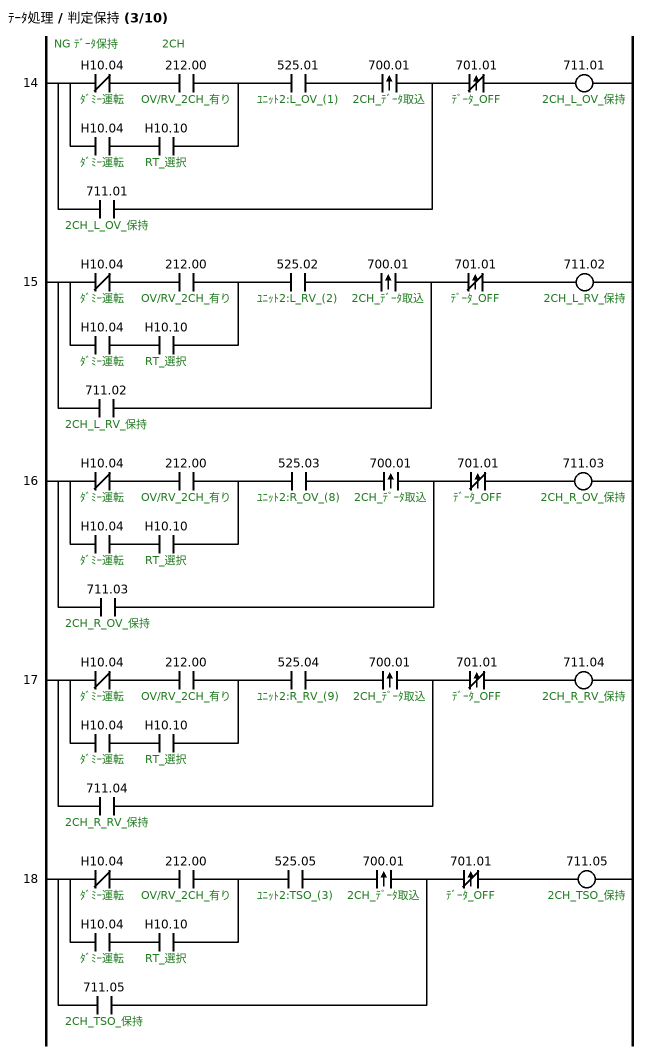
; [picture p144: ﾃｰﾀ処理 / 判定保持, rungs 14-18]
; rung 14: NG ﾃﾞｰﾀ保持　　　　2CH
LDNOT H10.04  ; ﾀﾞﾐｰ運転
AND 212.00  ; OV/RV_2CH_有り
LD H10.04  ; ﾀﾞﾐｰ運転
AND H10.10  ; RT_選択
ORLD
AND 525.01  ; ﾕﾆｯﾄ2:L_OV_(1)
@AND 700.01  ; 2CH_ﾃﾞｰﾀ取込
OR 711.01  ; 2CH_L_OV_保持
@ANDNOT 701.01  ; ﾃﾞｰﾀ_OFF
OUT 711.01  ; 2CH_L_OV_保持
; rung 15
LDNOT H10.04  ; ﾀﾞﾐｰ運転
AND 212.00  ; OV/RV_2CH_有り
LD H10.04  ; ﾀﾞﾐｰ運転
AND H10.10  ; RT_選択
ORLD
AND 525.02  ; ﾕﾆｯﾄ2:L_RV_(2)
@AND 700.01  ; 2CH_ﾃﾞｰﾀ取込
OR 711.02  ; 2CH_L_RV_保持
@ANDNOT 701.01  ; ﾃﾞｰﾀ_OFF
OUT 711.02  ; 2CH_L_RV_保持
; rung 16
LDNOT H10.04  ; ﾀﾞﾐｰ運転
AND 212.00  ; OV/RV_2CH_有り
LD H10.04  ; ﾀﾞﾐｰ運転
AND H10.10  ; RT_選択
ORLD
AND 525.03  ; ﾕﾆｯﾄ2:R_OV_(8)
@AND 700.01  ; 2CH_ﾃﾞｰﾀ取込
OR 711.03  ; 2CH_R_OV_保持
@ANDNOT 701.01  ; ﾃﾞｰﾀ_OFF
OUT 711.03  ; 2CH_R_OV_保持
; rung 17
LDNOT H10.04  ; ﾀﾞﾐｰ運転
AND 212.00  ; OV/RV_2CH_有り
LD H10.04  ; ﾀﾞﾐｰ運転
AND H10.10  ; RT_選択
ORLD
AND 525.04  ; ﾕﾆｯﾄ2:R_RV_(9)
@AND 700.01  ; 2CH_ﾃﾞｰﾀ取込
OR 711.04  ; 2CH_R_RV_保持
@ANDNOT 701.01  ; ﾃﾞｰﾀ_OFF
OUT 711.04  ; 2CH_R_RV_保持
; rung 18
LDNOT H10.04  ; ﾀﾞﾐｰ運転
AND 212.00  ; OV/RV_2CH_有り
LD H10.04  ; ﾀﾞﾐｰ運転
AND H10.10  ; RT_選択
ORLD
AND 525.05  ; ﾕﾆｯﾄ2:TSO_(3)
@AND 700.01  ; 2CH_ﾃﾞｰﾀ取込
OR 711.05  ; 2CH_TSO_保持
@ANDNOT 701.01  ; ﾃﾞｰﾀ_OFF
OUT 711.05  ; 2CH_TSO_保持

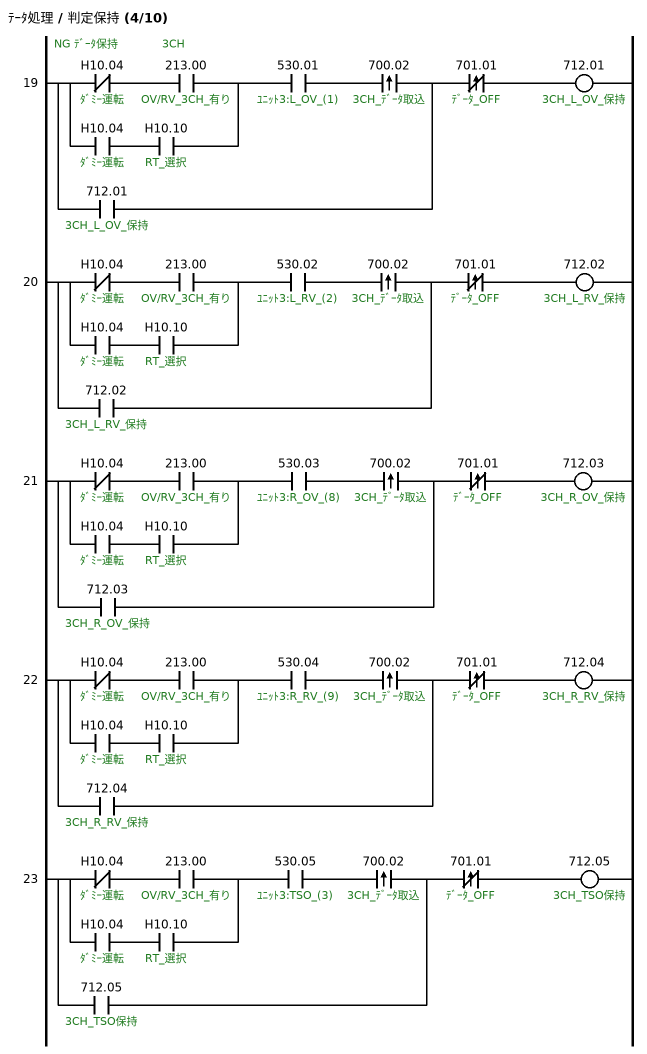
; rung 19: NG ﾃﾞｰﾀ保持　　　　3CH
LDNOT H10.04  ; ﾀﾞﾐｰ運転
AND 213.00  ; OV/RV_3CH_有り
LD H10.04  ; ﾀﾞﾐｰ運転
AND H10.10  ; RT_選択
ORLD
AND 530.01  ; ﾕﾆｯﾄ3:L_OV_(1)
@AND 700.02  ; 3CH_ﾃﾞｰﾀ取込
OR 712.01  ; 3CH_L_OV_保持
@ANDNOT 701.01  ; ﾃﾞｰﾀ_OFF
OUT 712.01  ; 3CH_L_OV_保持
; rung 20
LDNOT H10.04  ; ﾀﾞﾐｰ運転
AND 213.00  ; OV/RV_3CH_有り
LD H10.04  ; ﾀﾞﾐｰ運転
AND H10.10  ; RT_選択
ORLD
AND 530.02  ; ﾕﾆｯﾄ3:L_RV_(2)
@AND 700.02  ; 3CH_ﾃﾞｰﾀ取込
OR 712.02  ; 3CH_L_RV_保持
@ANDNOT 701.01  ; ﾃﾞｰﾀ_OFF
OUT 712.02  ; 3CH_L_RV_保持
; rung 21
LDNOT H10.04  ; ﾀﾞﾐｰ運転
AND 213.00  ; OV/RV_3CH_有り
LD H10.04  ; ﾀﾞﾐｰ運転
AND H10.10  ; RT_選択
ORLD
AND 530.03  ; ﾕﾆｯﾄ3:R_OV_(8)
@AND 700.02  ; 3CH_ﾃﾞｰﾀ取込
OR 712.03  ; 3CH_R_OV_保持
@ANDNOT 701.01  ; ﾃﾞｰﾀ_OFF
OUT 712.03  ; 3CH_R_OV_保持
; rung 22
LDNOT H10.04  ; ﾀﾞﾐｰ運転
AND 213.00  ; OV/RV_3CH_有り
LD H10.04  ; ﾀﾞﾐｰ運転
AND H10.10  ; RT_選択
ORLD
AND 530.04  ; ﾕﾆｯﾄ3:R_RV_(9)
@AND 700.02  ; 3CH_ﾃﾞｰﾀ取込
OR 712.04  ; 3CH_R_RV_保持
@ANDNOT 701.01  ; ﾃﾞｰﾀ_OFF
OUT 712.04  ; 3CH_R_RV_保持
; rung 23
LDNOT H10.04  ; ﾀﾞﾐｰ運転
AND 213.00  ; OV/RV_3CH_有り
LD H10.04  ; ﾀﾞﾐｰ運転
AND H10.10  ; RT_選択
ORLD
AND 530.05  ; ﾕﾆｯﾄ3:TSO_(3)
@AND 700.02  ; 3CH_ﾃﾞｰﾀ取込
OR 712.05  ; 3CH_TSO保持
@ANDNOT 701.01  ; ﾃﾞｰﾀ_OFF
OUT 712.05  ; 3CH_TSO保持

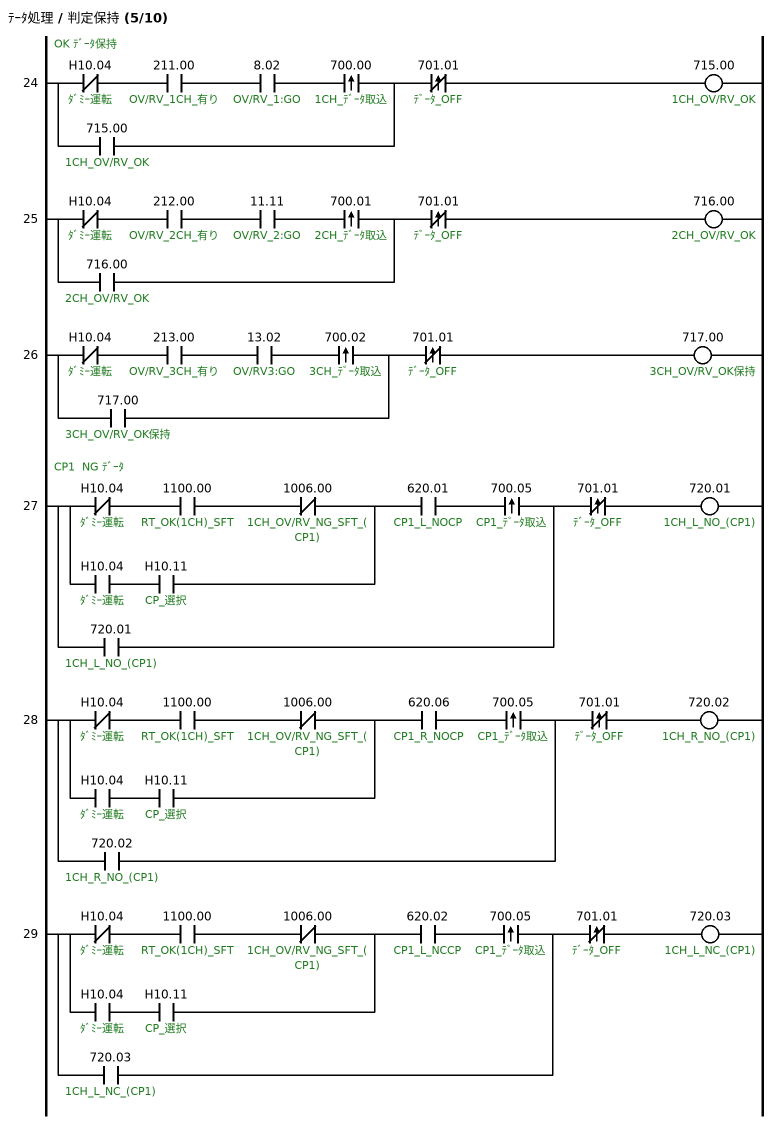
; rung 24: OK ﾃﾞｰﾀ保持
LDNOT H10.04  ; ﾀﾞﾐｰ運転
AND 211.00  ; OV/RV_1CH_有り
AND 8.02  ; OV/RV_1:GO
@AND 700.00  ; 1CH_ﾃﾞｰﾀ取込
OR 715.00  ; 1CH_OV/RV_OK
@ANDNOT 701.01  ; ﾃﾞｰﾀ_OFF
OUT 715.00  ; 1CH_OV/RV_OK
; rung 25
LDNOT H10.04  ; ﾀﾞﾐｰ運転
AND 212.00  ; OV/RV_2CH_有り
AND 11.11  ; OV/RV_2:GO
@AND 700.01  ; 2CH_ﾃﾞｰﾀ取込
OR 716.00  ; 2CH_OV/RV_OK
@ANDNOT 701.01  ; ﾃﾞｰﾀ_OFF
OUT 716.00  ; 2CH_OV/RV_OK
; rung 26
LDNOT H10.04  ; ﾀﾞﾐｰ運転
AND 213.00  ; OV/RV_3CH_有り
AND 13.02  ; OV/RV3:GO
@AND 700.02  ; 3CH_ﾃﾞｰﾀ取込
OR 717.00  ; 3CH_OV/RV_OK保持
@ANDNOT 701.01  ; ﾃﾞｰﾀ_OFF
OUT 717.00  ; 3CH_OV/RV_OK保持
; rung 27: CP1  NG ﾃﾞｰﾀ
LDNOT H10.04  ; ﾀﾞﾐｰ運転
AND 1100.00  ; RT_OK(1CH)_SFT
ANDNOT 1006.00  ; 1CH_OV/RV_NG_SFT_(CP1)
LD H10.04  ; ﾀﾞﾐｰ運転
AND H10.11  ; CP_選択
ORLD
AND 620.01  ; CP1_L_NOCP
@AND 700.05  ; CP1_ﾃﾞｰﾀ取込
OR 720.01  ; 1CH_L_NO_(CP1)
@ANDNOT 701.01  ; ﾃﾞｰﾀ_OFF
OUT 720.01  ; 1CH_L_NO_(CP1)
; rung 28
LDNOT H10.04  ; ﾀﾞﾐｰ運転
AND 1100.00  ; RT_OK(1CH)_SFT
ANDNOT 1006.00  ; 1CH_OV/RV_NG_SFT_(CP1)
LD H10.04  ; ﾀﾞﾐｰ運転
AND H10.11  ; CP_選択
ORLD
AND 620.06  ; CP1_R_NOCP
@AND 700.05  ; CP1_ﾃﾞｰﾀ取込
OR 720.02  ; 1CH_R_NO_(CP1)
@ANDNOT 701.01  ; ﾃﾞｰﾀ_OFF
OUT 720.02  ; 1CH_R_NO_(CP1)
; rung 29
LDNOT H10.04  ; ﾀﾞﾐｰ運転
AND 1100.00  ; RT_OK(1CH)_SFT
ANDNOT 1006.00  ; 1CH_OV/RV_NG_SFT_(CP1)
LD H10.04  ; ﾀﾞﾐｰ運転
AND H10.11  ; CP_選択
ORLD
AND 620.02  ; CP1_L_NCCP
@AND 700.05  ; CP1_ﾃﾞｰﾀ取込
OR 720.03  ; 1CH_L_NC_(CP1)
@ANDNOT 701.01  ; ﾃﾞｰﾀ_OFF
OUT 720.03  ; 1CH_L_NC_(CP1)

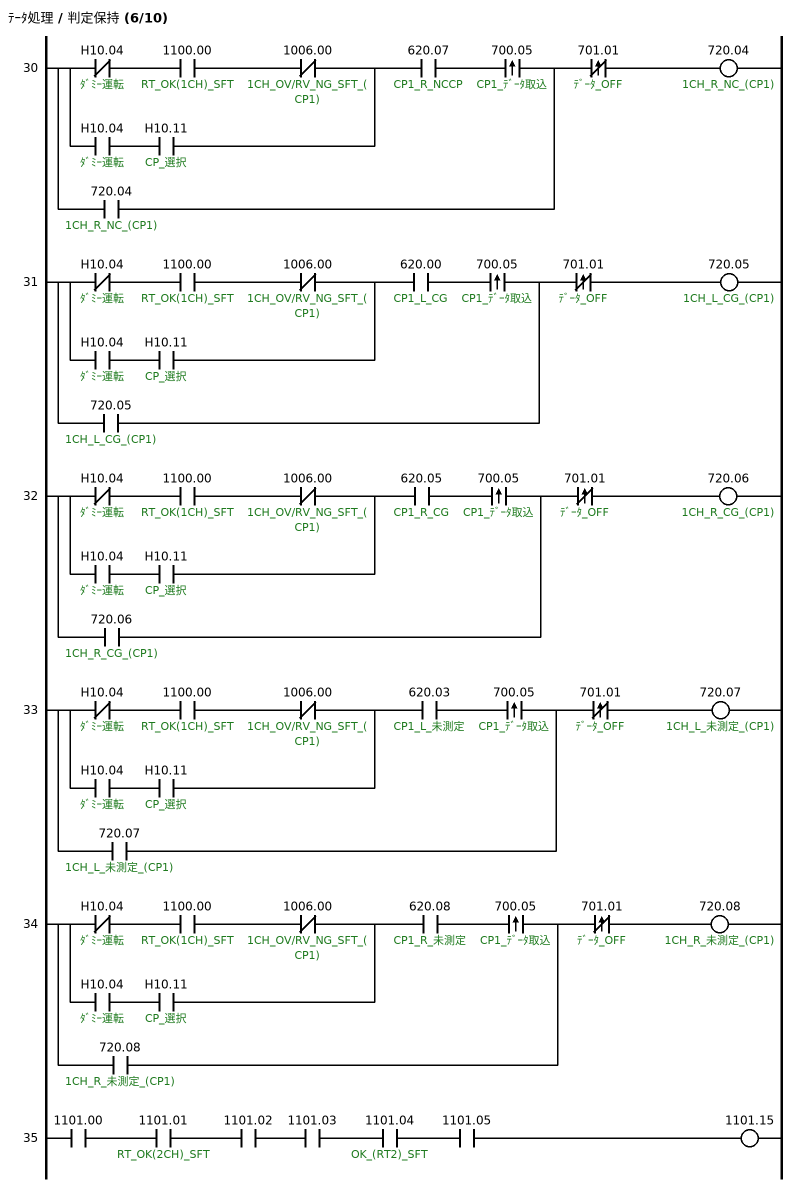
; rung 30
LDNOT H10.04  ; ﾀﾞﾐｰ運転
AND 1100.00  ; RT_OK(1CH)_SFT
ANDNOT 1006.00  ; 1CH_OV/RV_NG_SFT_(CP1)
LD H10.04  ; ﾀﾞﾐｰ運転
AND H10.11  ; CP_選択
ORLD
AND 620.07  ; CP1_R_NCCP
@AND 700.05  ; CP1_ﾃﾞｰﾀ取込
OR 720.04  ; 1CH_R_NC_(CP1)
@ANDNOT 701.01  ; ﾃﾞｰﾀ_OFF
OUT 720.04  ; 1CH_R_NC_(CP1)
; rung 31
LDNOT H10.04  ; ﾀﾞﾐｰ運転
AND 1100.00  ; RT_OK(1CH)_SFT
ANDNOT 1006.00  ; 1CH_OV/RV_NG_SFT_(CP1)
LD H10.04  ; ﾀﾞﾐｰ運転
AND H10.11  ; CP_選択
ORLD
AND 620.00  ; CP1_L_CG
@AND 700.05  ; CP1_ﾃﾞｰﾀ取込
OR 720.05  ; 1CH_L_CG_(CP1)
@ANDNOT 701.01  ; ﾃﾞｰﾀ_OFF
OUT 720.05  ; 1CH_L_CG_(CP1)
; rung 32
LDNOT H10.04  ; ﾀﾞﾐｰ運転
AND 1100.00  ; RT_OK(1CH)_SFT
ANDNOT 1006.00  ; 1CH_OV/RV_NG_SFT_(CP1)
LD H10.04  ; ﾀﾞﾐｰ運転
AND H10.11  ; CP_選択
ORLD
AND 620.05  ; CP1_R_CG
@AND 700.05  ; CP1_ﾃﾞｰﾀ取込
OR 720.06  ; 1CH_R_CG_(CP1)
@ANDNOT 701.01  ; ﾃﾞｰﾀ_OFF
OUT 720.06  ; 1CH_R_CG_(CP1)
; rung 33
LDNOT H10.04  ; ﾀﾞﾐｰ運転
AND 1100.00  ; RT_OK(1CH)_SFT
ANDNOT 1006.00  ; 1CH_OV/RV_NG_SFT_(CP1)
LD H10.04  ; ﾀﾞﾐｰ運転
AND H10.11  ; CP_選択
ORLD
AND 620.03  ; CP1_L_未測定
@AND 700.05  ; CP1_ﾃﾞｰﾀ取込
OR 720.07  ; 1CH_L_未測定_(CP1)
@ANDNOT 701.01  ; ﾃﾞｰﾀ_OFF
OUT 720.07  ; 1CH_L_未測定_(CP1)
; rung 34
LDNOT H10.04  ; ﾀﾞﾐｰ運転
AND 1100.00  ; RT_OK(1CH)_SFT
ANDNOT 1006.00  ; 1CH_OV/RV_NG_SFT_(CP1)
LD H10.04  ; ﾀﾞﾐｰ運転
AND H10.11  ; CP_選択
ORLD
AND 620.08  ; CP1_R_未測定
@AND 700.05  ; CP1_ﾃﾞｰﾀ取込
OR 720.08  ; 1CH_R_未測定_(CP1)
@ANDNOT 701.01  ; ﾃﾞｰﾀ_OFF
OUT 720.08  ; 1CH_R_未測定_(CP1)
; rung 35
LD 1101.00
AND 1101.01  ; RT_OK(2CH)_SFT
AND 1101.02
AND 1101.03
AND 1101.04  ; OK_(RT2)_SFT
AND 1101.05
OUT 1101.15

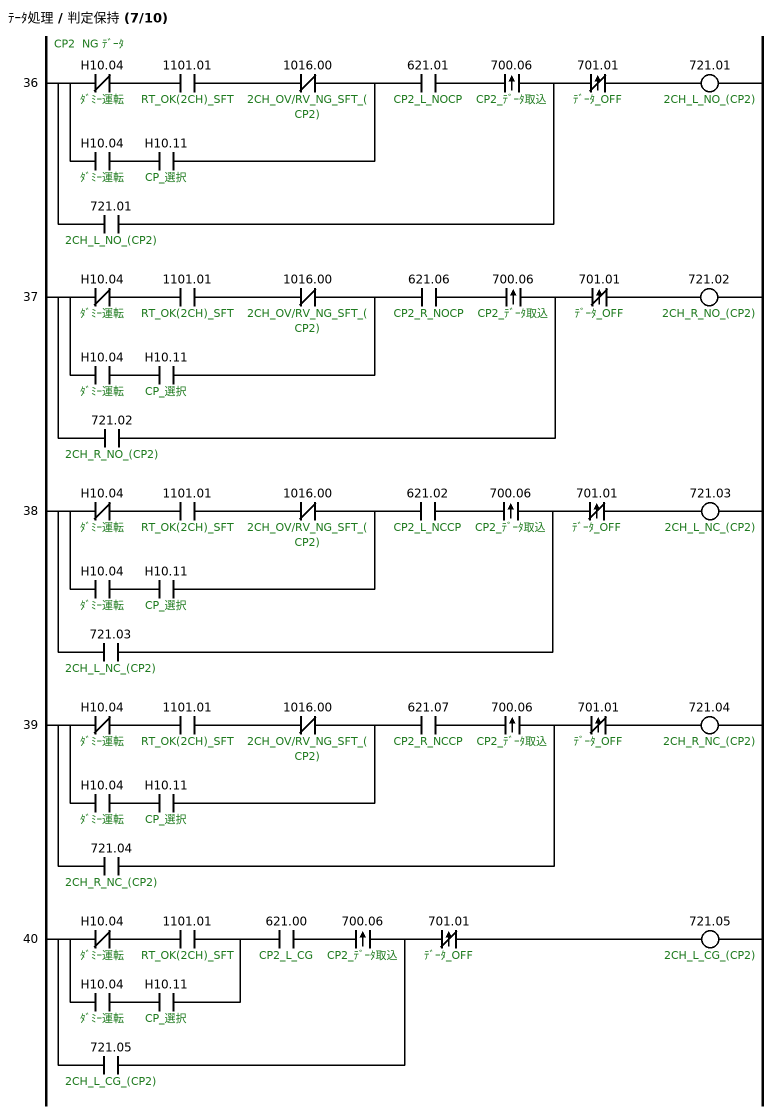
; rung 36: CP2  NG ﾃﾞｰﾀ
LDNOT H10.04  ; ﾀﾞﾐｰ運転
AND 1101.01  ; RT_OK(2CH)_SFT
ANDNOT 1016.00  ; 2CH_OV/RV_NG_SFT_(CP2)
LD H10.04  ; ﾀﾞﾐｰ運転
AND H10.11  ; CP_選択
ORLD
AND 621.01  ; CP2_L_NOCP
@AND 700.06  ; CP2_ﾃﾞｰﾀ取込
OR 721.01  ; 2CH_L_NO_(CP2)
@ANDNOT 701.01  ; ﾃﾞｰﾀ_OFF
OUT 721.01  ; 2CH_L_NO_(CP2)
; rung 37
LDNOT H10.04  ; ﾀﾞﾐｰ運転
AND 1101.01  ; RT_OK(2CH)_SFT
ANDNOT 1016.00  ; 2CH_OV/RV_NG_SFT_(CP2)
LD H10.04  ; ﾀﾞﾐｰ運転
AND H10.11  ; CP_選択
ORLD
AND 621.06  ; CP2_R_NOCP
@AND 700.06  ; CP2_ﾃﾞｰﾀ取込
OR 721.02  ; 2CH_R_NO_(CP2)
@ANDNOT 701.01  ; ﾃﾞｰﾀ_OFF
OUT 721.02  ; 2CH_R_NO_(CP2)
; rung 38
LDNOT H10.04  ; ﾀﾞﾐｰ運転
AND 1101.01  ; RT_OK(2CH)_SFT
ANDNOT 1016.00  ; 2CH_OV/RV_NG_SFT_(CP2)
LD H10.04  ; ﾀﾞﾐｰ運転
AND H10.11  ; CP_選択
ORLD
AND 621.02  ; CP2_L_NCCP
@AND 700.06  ; CP2_ﾃﾞｰﾀ取込
OR 721.03  ; 2CH_L_NC_(CP2)
@ANDNOT 701.01  ; ﾃﾞｰﾀ_OFF
OUT 721.03  ; 2CH_L_NC_(CP2)
; rung 39
LDNOT H10.04  ; ﾀﾞﾐｰ運転
AND 1101.01  ; RT_OK(2CH)_SFT
ANDNOT 1016.00  ; 2CH_OV/RV_NG_SFT_(CP2)
LD H10.04  ; ﾀﾞﾐｰ運転
AND H10.11  ; CP_選択
ORLD
AND 621.07  ; CP2_R_NCCP
@AND 700.06  ; CP2_ﾃﾞｰﾀ取込
OR 721.04  ; 2CH_R_NC_(CP2)
@ANDNOT 701.01  ; ﾃﾞｰﾀ_OFF
OUT 721.04  ; 2CH_R_NC_(CP2)
; rung 40
LDNOT H10.04  ; ﾀﾞﾐｰ運転
AND 1101.01  ; RT_OK(2CH)_SFT
LD H10.04  ; ﾀﾞﾐｰ運転
AND H10.11  ; CP_選択
ORLD
AND 621.00  ; CP2_L_CG
@AND 700.06  ; CP2_ﾃﾞｰﾀ取込
OR 721.05  ; 2CH_L_CG_(CP2)
@ANDNOT 701.01  ; ﾃﾞｰﾀ_OFF
OUT 721.05  ; 2CH_L_CG_(CP2)

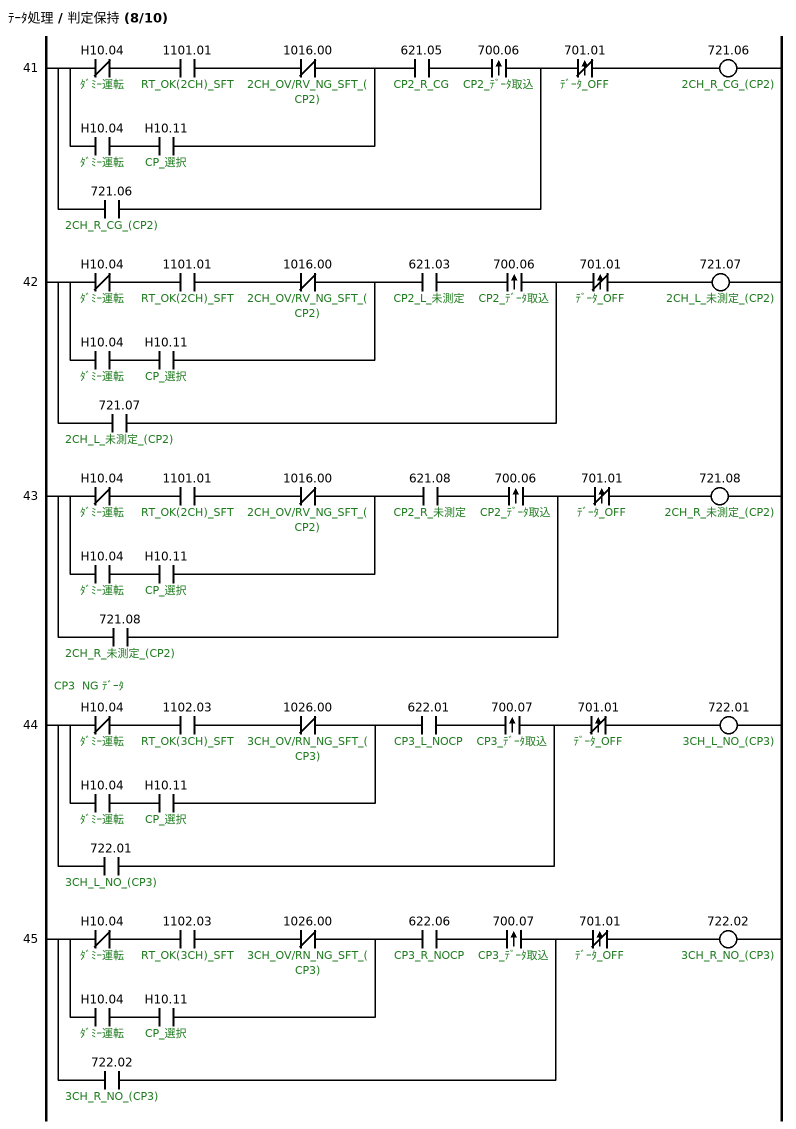
; rung 41
LDNOT H10.04  ; ﾀﾞﾐｰ運転
AND 1101.01  ; RT_OK(2CH)_SFT
ANDNOT 1016.00  ; 2CH_OV/RV_NG_SFT_(CP2)
LD H10.04  ; ﾀﾞﾐｰ運転
AND H10.11  ; CP_選択
ORLD
AND 621.05  ; CP2_R_CG
@AND 700.06  ; CP2_ﾃﾞｰﾀ取込
OR 721.06  ; 2CH_R_CG_(CP2)
@ANDNOT 701.01  ; ﾃﾞｰﾀ_OFF
OUT 721.06  ; 2CH_R_CG_(CP2)
; rung 42
LDNOT H10.04  ; ﾀﾞﾐｰ運転
AND 1101.01  ; RT_OK(2CH)_SFT
ANDNOT 1016.00  ; 2CH_OV/RV_NG_SFT_(CP2)
LD H10.04  ; ﾀﾞﾐｰ運転
AND H10.11  ; CP_選択
ORLD
AND 621.03  ; CP2_L_未測定
@AND 700.06  ; CP2_ﾃﾞｰﾀ取込
OR 721.07  ; 2CH_L_未測定_(CP2)
@ANDNOT 701.01  ; ﾃﾞｰﾀ_OFF
OUT 721.07  ; 2CH_L_未測定_(CP2)
; rung 43
LDNOT H10.04  ; ﾀﾞﾐｰ運転
AND 1101.01  ; RT_OK(2CH)_SFT
ANDNOT 1016.00  ; 2CH_OV/RV_NG_SFT_(CP2)
LD H10.04  ; ﾀﾞﾐｰ運転
AND H10.11  ; CP_選択
ORLD
AND 621.08  ; CP2_R_未測定
@AND 700.06  ; CP2_ﾃﾞｰﾀ取込
OR 721.08  ; 2CH_R_未測定_(CP2)
@ANDNOT 701.01  ; ﾃﾞｰﾀ_OFF
OUT 721.08  ; 2CH_R_未測定_(CP2)
; rung 44: CP3  NG ﾃﾞｰﾀ
LDNOT H10.04  ; ﾀﾞﾐｰ運転
AND 1102.03  ; RT_OK(3CH)_SFT
ANDNOT 1026.00  ; 3CH_OV/RN_NG_SFT_(CP3)
LD H10.04  ; ﾀﾞﾐｰ運転
AND H10.11  ; CP_選択
ORLD
AND 622.01  ; CP3_L_NOCP
@AND 700.07  ; CP3_ﾃﾞｰﾀ取込
OR 722.01  ; 3CH_L_NO_(CP3)
@ANDNOT 701.01  ; ﾃﾞｰﾀ_OFF
OUT 722.01  ; 3CH_L_NO_(CP3)
; rung 45
LDNOT H10.04  ; ﾀﾞﾐｰ運転
AND 1102.03  ; RT_OK(3CH)_SFT
ANDNOT 1026.00  ; 3CH_OV/RN_NG_SFT_(CP3)
LD H10.04  ; ﾀﾞﾐｰ運転
AND H10.11  ; CP_選択
ORLD
AND 622.06  ; CP3_R_NOCP
@AND 700.07  ; CP3_ﾃﾞｰﾀ取込
OR 722.02  ; 3CH_R_NO_(CP3)
@ANDNOT 701.01  ; ﾃﾞｰﾀ_OFF
OUT 722.02  ; 3CH_R_NO_(CP3)

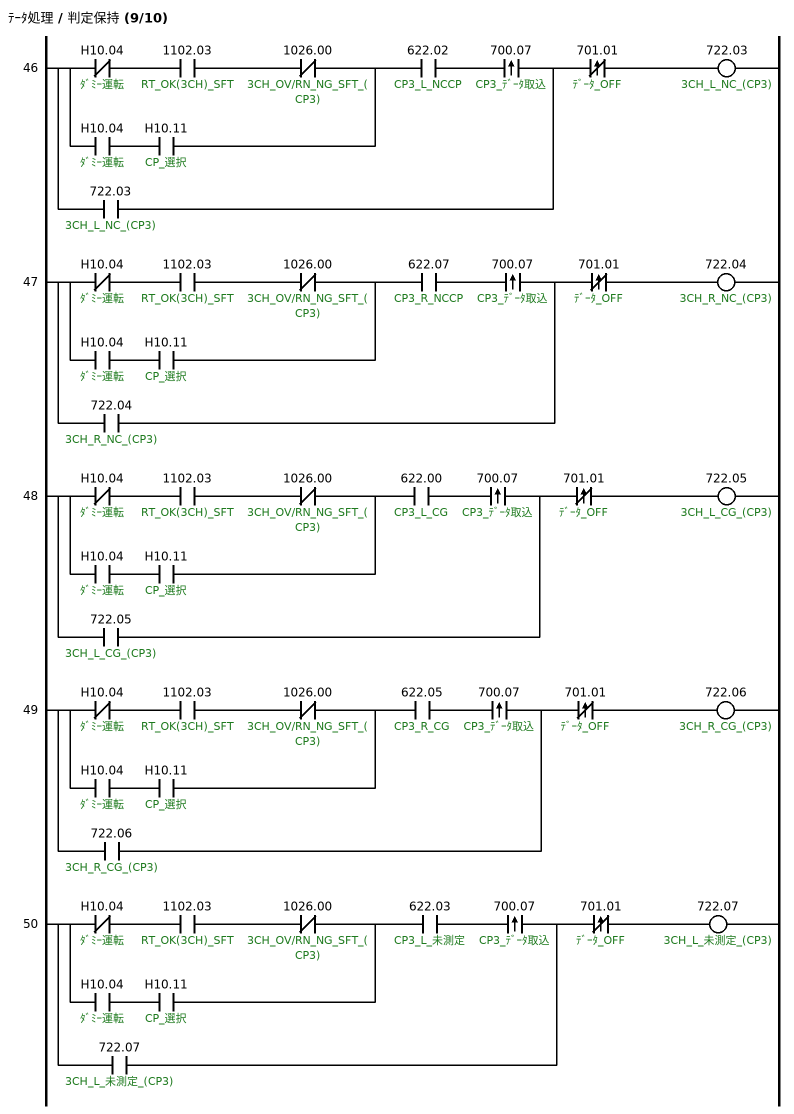
; rung 46
LDNOT H10.04  ; ﾀﾞﾐｰ運転
AND 1102.03  ; RT_OK(3CH)_SFT
ANDNOT 1026.00  ; 3CH_OV/RN_NG_SFT_(CP3)
LD H10.04  ; ﾀﾞﾐｰ運転
AND H10.11  ; CP_選択
ORLD
AND 622.02  ; CP3_L_NCCP
@AND 700.07  ; CP3_ﾃﾞｰﾀ取込
OR 722.03  ; 3CH_L_NC_(CP3)
@ANDNOT 701.01  ; ﾃﾞｰﾀ_OFF
OUT 722.03  ; 3CH_L_NC_(CP3)
; rung 47
LDNOT H10.04  ; ﾀﾞﾐｰ運転
AND 1102.03  ; RT_OK(3CH)_SFT
ANDNOT 1026.00  ; 3CH_OV/RN_NG_SFT_(CP3)
LD H10.04  ; ﾀﾞﾐｰ運転
AND H10.11  ; CP_選択
ORLD
AND 622.07  ; CP3_R_NCCP
@AND 700.07  ; CP3_ﾃﾞｰﾀ取込
OR 722.04  ; 3CH_R_NC_(CP3)
@ANDNOT 701.01  ; ﾃﾞｰﾀ_OFF
OUT 722.04  ; 3CH_R_NC_(CP3)
; rung 48
LDNOT H10.04  ; ﾀﾞﾐｰ運転
AND 1102.03  ; RT_OK(3CH)_SFT
ANDNOT 1026.00  ; 3CH_OV/RN_NG_SFT_(CP3)
LD H10.04  ; ﾀﾞﾐｰ運転
AND H10.11  ; CP_選択
ORLD
AND 622.00  ; CP3_L_CG
@AND 700.07  ; CP3_ﾃﾞｰﾀ取込
OR 722.05  ; 3CH_L_CG_(CP3)
@ANDNOT 701.01  ; ﾃﾞｰﾀ_OFF
OUT 722.05  ; 3CH_L_CG_(CP3)
; rung 49
LDNOT H10.04  ; ﾀﾞﾐｰ運転
AND 1102.03  ; RT_OK(3CH)_SFT
ANDNOT 1026.00  ; 3CH_OV/RN_NG_SFT_(CP3)
LD H10.04  ; ﾀﾞﾐｰ運転
AND H10.11  ; CP_選択
ORLD
AND 622.05  ; CP3_R_CG
@AND 700.07  ; CP3_ﾃﾞｰﾀ取込
OR 722.06  ; 3CH_R_CG_(CP3)
@ANDNOT 701.01  ; ﾃﾞｰﾀ_OFF
OUT 722.06  ; 3CH_R_CG_(CP3)
; rung 50
LDNOT H10.04  ; ﾀﾞﾐｰ運転
AND 1102.03  ; RT_OK(3CH)_SFT
ANDNOT 1026.00  ; 3CH_OV/RN_NG_SFT_(CP3)
LD H10.04  ; ﾀﾞﾐｰ運転
AND H10.11  ; CP_選択
ORLD
AND 622.03  ; CP3_L_未測定
@AND 700.07  ; CP3_ﾃﾞｰﾀ取込
OR 722.07  ; 3CH_L_未測定_(CP3)
@ANDNOT 701.01  ; ﾃﾞｰﾀ_OFF
OUT 722.07  ; 3CH_L_未測定_(CP3)

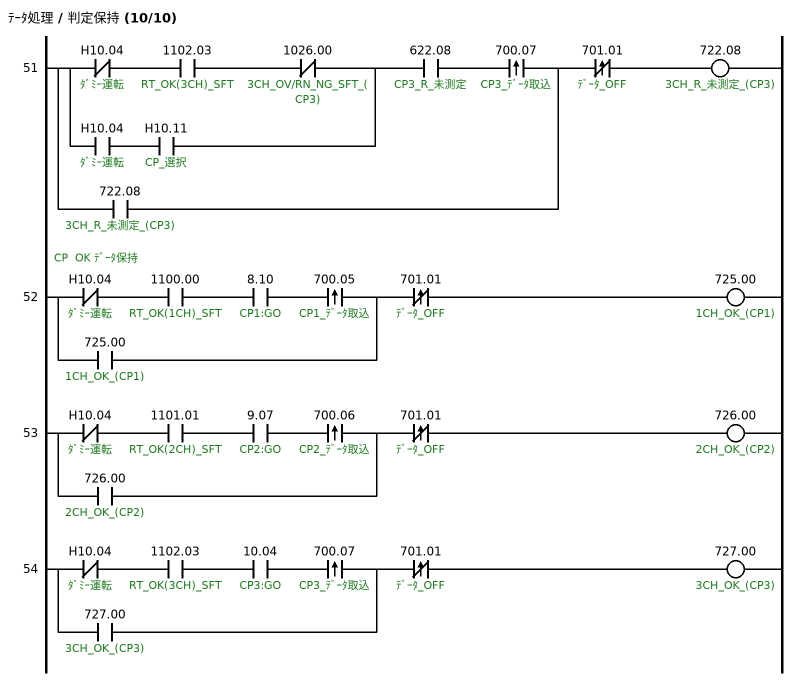
; rung 51
LDNOT H10.04  ; ﾀﾞﾐｰ運転
AND 1102.03  ; RT_OK(3CH)_SFT
ANDNOT 1026.00  ; 3CH_OV/RN_NG_SFT_(CP3)
LD H10.04  ; ﾀﾞﾐｰ運転
AND H10.11  ; CP_選択
ORLD
AND 622.08  ; CP3_R_未測定
@AND 700.07  ; CP3_ﾃﾞｰﾀ取込
OR 722.08  ; 3CH_R_未測定_(CP3)
@ANDNOT 701.01  ; ﾃﾞｰﾀ_OFF
OUT 722.08  ; 3CH_R_未測定_(CP3)
; rung 52: CP  OK ﾃﾞｰﾀ保持
LDNOT H10.04  ; ﾀﾞﾐｰ運転
AND 1100.00  ; RT_OK(1CH)_SFT
AND 8.10  ; CP1:GO
@AND 700.05  ; CP1_ﾃﾞｰﾀ取込
OR 725.00  ; 1CH_OK_(CP1)
@ANDNOT 701.01  ; ﾃﾞｰﾀ_OFF
OUT 725.00  ; 1CH_OK_(CP1)
; rung 53
LDNOT H10.04  ; ﾀﾞﾐｰ運転
AND 1101.01  ; RT_OK(2CH)_SFT
AND 9.07  ; CP2:GO
@AND 700.06  ; CP2_ﾃﾞｰﾀ取込
OR 726.00  ; 2CH_OK_(CP2)
@ANDNOT 701.01  ; ﾃﾞｰﾀ_OFF
OUT 726.00  ; 2CH_OK_(CP2)
; rung 54
LDNOT H10.04  ; ﾀﾞﾐｰ運転
AND 1102.03  ; RT_OK(3CH)_SFT
AND 10.04  ; CP3:GO
@AND 700.07  ; CP3_ﾃﾞｰﾀ取込
OR 727.00  ; 3CH_OK_(CP3)
@ANDNOT 701.01  ; ﾃﾞｰﾀ_OFF
OUT 727.00  ; 3CH_OK_(CP3)

### Section NG_SFT

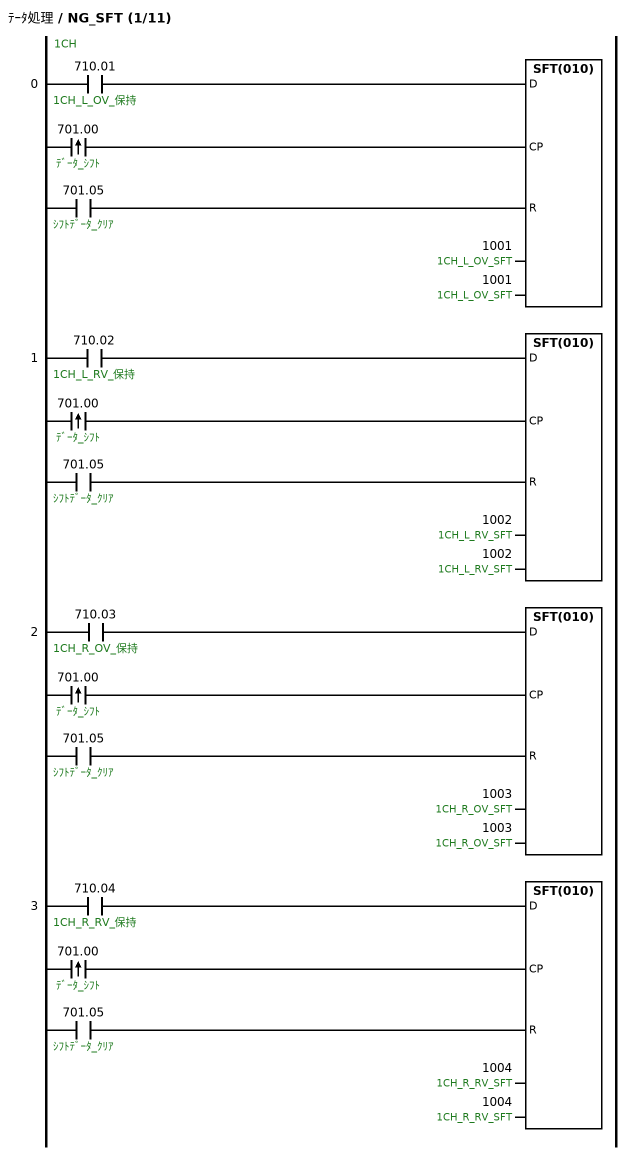
; rung 0: 1CH
LD 710.01  ; 1CH_L_OV_保持
@LD 701.00  ; ﾃﾞｰﾀ_ｼﾌﾄ
LD 701.05  ; ｼﾌﾄﾃﾞｰﾀ_ｸﾘｱ
SFT(010) 1001 1001  ; 1CH_L_OV_SFT
; rung 1
LD 710.02  ; 1CH_L_RV_保持
@LD 701.00  ; ﾃﾞｰﾀ_ｼﾌﾄ
LD 701.05  ; ｼﾌﾄﾃﾞｰﾀ_ｸﾘｱ
SFT(010) 1002 1002  ; 1CH_L_RV_SFT
; rung 2
LD 710.03  ; 1CH_R_OV_保持
@LD 701.00  ; ﾃﾞｰﾀ_ｼﾌﾄ
LD 701.05  ; ｼﾌﾄﾃﾞｰﾀ_ｸﾘｱ
SFT(010) 1003 1003  ; 1CH_R_OV_SFT
; rung 3
LD 710.04  ; 1CH_R_RV_保持
@LD 701.00  ; ﾃﾞｰﾀ_ｼﾌﾄ
LD 701.05  ; ｼﾌﾄﾃﾞｰﾀ_ｸﾘｱ
SFT(010) 1004 1004  ; 1CH_R_RV_SFT

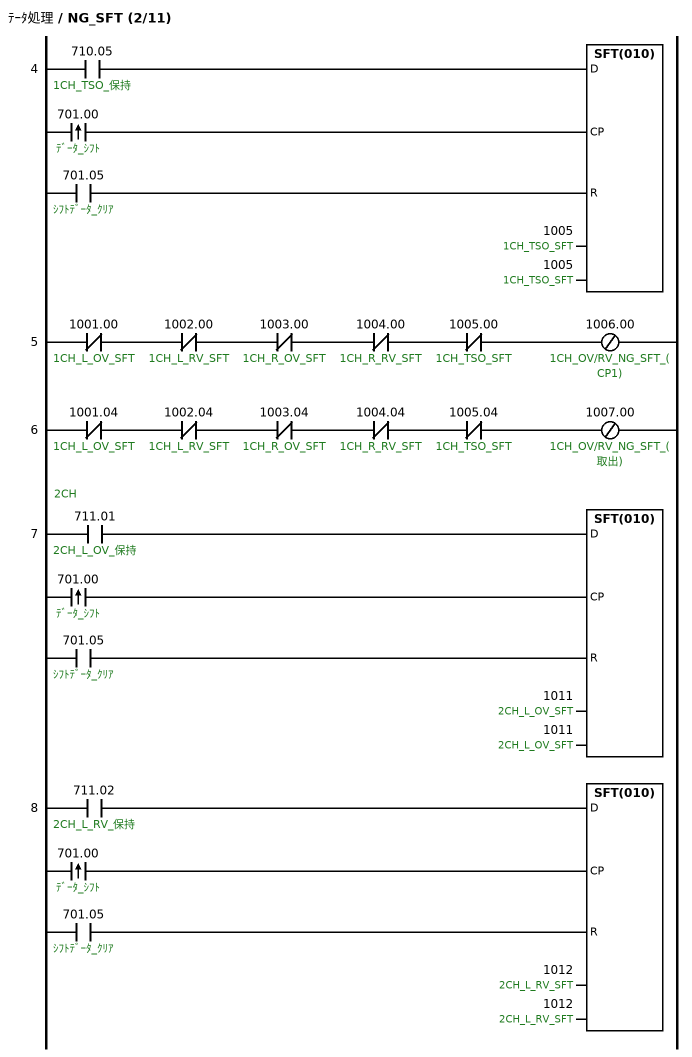
; rung 4
LD 710.05  ; 1CH_TSO_保持
@LD 701.00  ; ﾃﾞｰﾀ_ｼﾌﾄ
LD 701.05  ; ｼﾌﾄﾃﾞｰﾀ_ｸﾘｱ
SFT(010) 1005 1005  ; 1CH_TSO_SFT
; rung 5
LDNOT 1001.00  ; 1CH_L_OV_SFT
ANDNOT 1002.00  ; 1CH_L_RV_SFT
ANDNOT 1003.00  ; 1CH_R_OV_SFT
ANDNOT 1004.00  ; 1CH_R_RV_SFT
ANDNOT 1005.00  ; 1CH_TSO_SFT
OUTNOT 1006.00  ; 1CH_OV/RV_NG_SFT_(CP1)
; rung 6
LDNOT 1001.04  ; 1CH_L_OV_SFT
ANDNOT 1002.04  ; 1CH_L_RV_SFT
ANDNOT 1003.04  ; 1CH_R_OV_SFT
ANDNOT 1004.04  ; 1CH_R_RV_SFT
ANDNOT 1005.04  ; 1CH_TSO_SFT
OUTNOT 1007.00  ; 1CH_OV/RV_NG_SFT_(取出)
; rung 7: 2CH
LD 711.01  ; 2CH_L_OV_保持
@LD 701.00  ; ﾃﾞｰﾀ_ｼﾌﾄ
LD 701.05  ; ｼﾌﾄﾃﾞｰﾀ_ｸﾘｱ
SFT(010) 1011 1011  ; 2CH_L_OV_SFT
; rung 8
LD 711.02  ; 2CH_L_RV_保持
@LD 701.00  ; ﾃﾞｰﾀ_ｼﾌﾄ
LD 701.05  ; ｼﾌﾄﾃﾞｰﾀ_ｸﾘｱ
SFT(010) 1012 1012  ; 2CH_L_RV_SFT

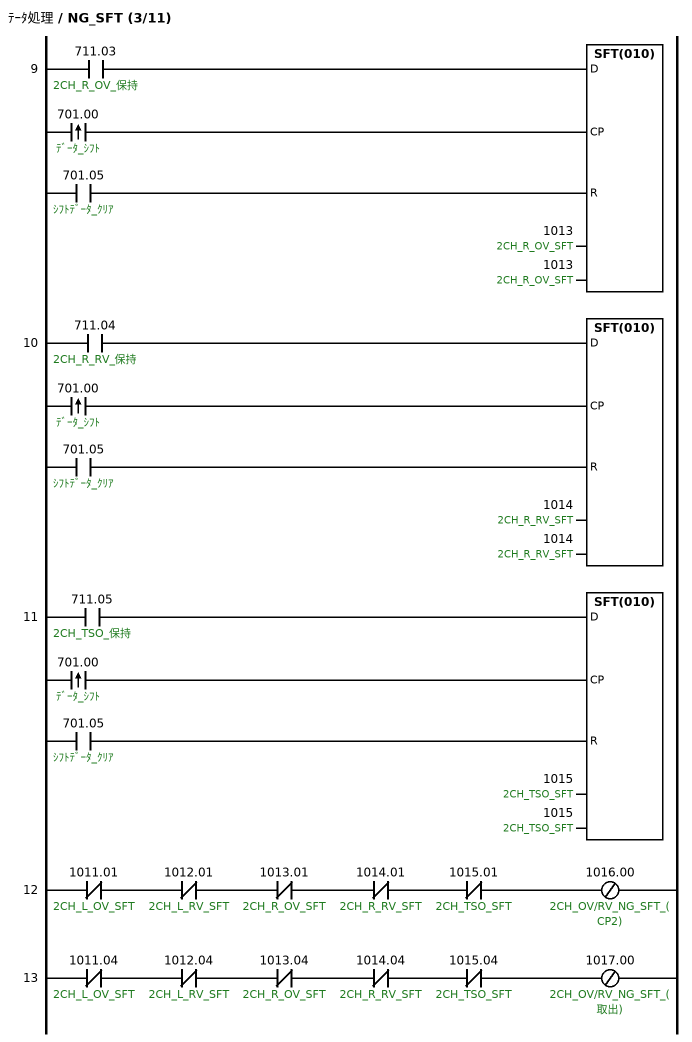
; rung 9
LD 711.03  ; 2CH_R_OV_保持
@LD 701.00  ; ﾃﾞｰﾀ_ｼﾌﾄ
LD 701.05  ; ｼﾌﾄﾃﾞｰﾀ_ｸﾘｱ
SFT(010) 1013 1013  ; 2CH_R_OV_SFT
; rung 10
LD 711.04  ; 2CH_R_RV_保持
@LD 701.00  ; ﾃﾞｰﾀ_ｼﾌﾄ
LD 701.05  ; ｼﾌﾄﾃﾞｰﾀ_ｸﾘｱ
SFT(010) 1014 1014  ; 2CH_R_RV_SFT
; rung 11
LD 711.05  ; 2CH_TSO_保持
@LD 701.00  ; ﾃﾞｰﾀ_ｼﾌﾄ
LD 701.05  ; ｼﾌﾄﾃﾞｰﾀ_ｸﾘｱ
SFT(010) 1015 1015  ; 2CH_TSO_SFT
; rung 12
LDNOT 1011.01  ; 2CH_L_OV_SFT
ANDNOT 1012.01  ; 2CH_L_RV_SFT
ANDNOT 1013.01  ; 2CH_R_OV_SFT
ANDNOT 1014.01  ; 2CH_R_RV_SFT
ANDNOT 1015.01  ; 2CH_TSO_SFT
OUTNOT 1016.00  ; 2CH_OV/RV_NG_SFT_(CP2)
; rung 13
LDNOT 1011.04  ; 2CH_L_OV_SFT
ANDNOT 1012.04  ; 2CH_L_RV_SFT
ANDNOT 1013.04  ; 2CH_R_OV_SFT
ANDNOT 1014.04  ; 2CH_R_RV_SFT
ANDNOT 1015.04  ; 2CH_TSO_SFT
OUTNOT 1017.00  ; 2CH_OV/RV_NG_SFT_(取出)

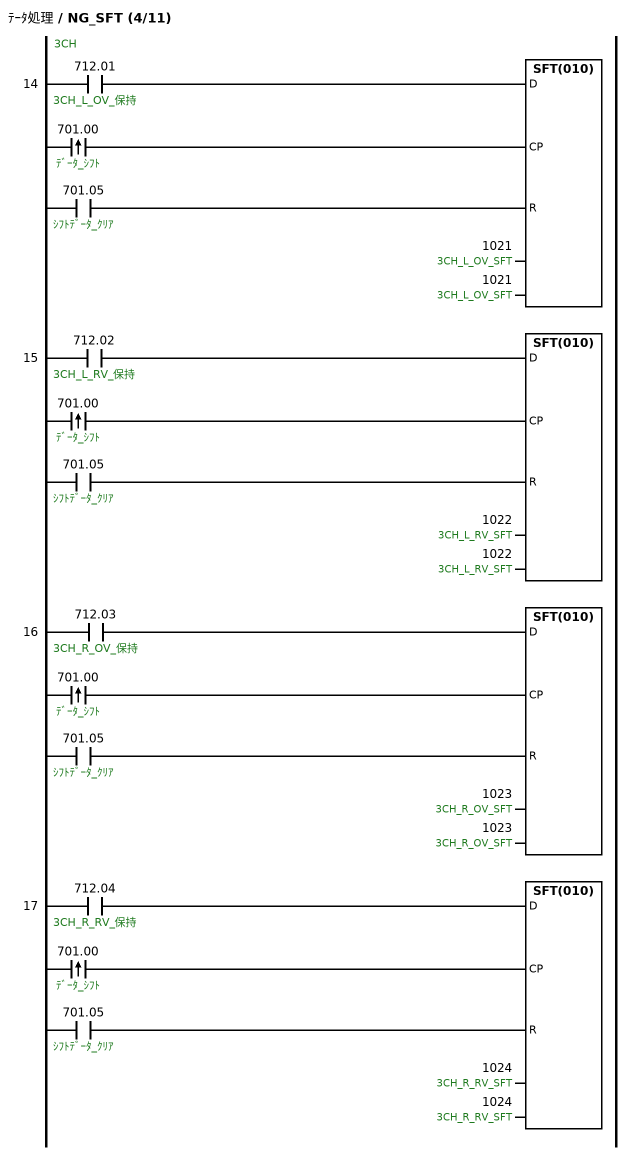
; rung 14: 3CH
LD 712.01  ; 3CH_L_OV_保持
@LD 701.00  ; ﾃﾞｰﾀ_ｼﾌﾄ
LD 701.05  ; ｼﾌﾄﾃﾞｰﾀ_ｸﾘｱ
SFT(010) 1021 1021  ; 3CH_L_OV_SFT
; rung 15
LD 712.02  ; 3CH_L_RV_保持
@LD 701.00  ; ﾃﾞｰﾀ_ｼﾌﾄ
LD 701.05  ; ｼﾌﾄﾃﾞｰﾀ_ｸﾘｱ
SFT(010) 1022 1022  ; 3CH_L_RV_SFT
; rung 16
LD 712.03  ; 3CH_R_OV_保持
@LD 701.00  ; ﾃﾞｰﾀ_ｼﾌﾄ
LD 701.05  ; ｼﾌﾄﾃﾞｰﾀ_ｸﾘｱ
SFT(010) 1023 1023  ; 3CH_R_OV_SFT
; rung 17
LD 712.04  ; 3CH_R_RV_保持
@LD 701.00  ; ﾃﾞｰﾀ_ｼﾌﾄ
LD 701.05  ; ｼﾌﾄﾃﾞｰﾀ_ｸﾘｱ
SFT(010) 1024 1024  ; 3CH_R_RV_SFT

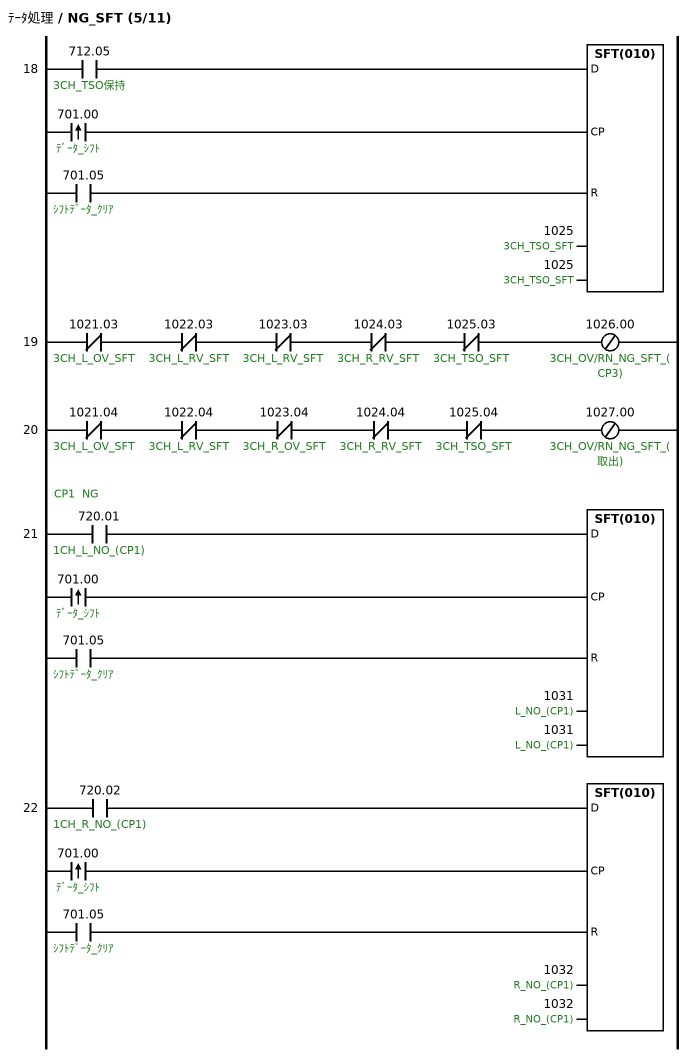
; rung 18
LD 712.05  ; 3CH_TSO保持
@LD 701.00  ; ﾃﾞｰﾀ_ｼﾌﾄ
LD 701.05  ; ｼﾌﾄﾃﾞｰﾀ_ｸﾘｱ
SFT(010) 1025 1025  ; 3CH_TSO_SFT
; rung 19
LDNOT 1021.03  ; 3CH_L_OV_SFT
ANDNOT 1022.03  ; 3CH_L_RV_SFT
ANDNOT 1023.03  ; 3CH_L_RV_SFT
ANDNOT 1024.03  ; 3CH_R_RV_SFT
ANDNOT 1025.03  ; 3CH_TSO_SFT
OUTNOT 1026.00  ; 3CH_OV/RN_NG_SFT_(CP3)
; rung 20
LDNOT 1021.04  ; 3CH_L_OV_SFT
ANDNOT 1022.04  ; 3CH_L_RV_SFT
ANDNOT 1023.04  ; 3CH_R_OV_SFT
ANDNOT 1024.04  ; 3CH_R_RV_SFT
ANDNOT 1025.04  ; 3CH_TSO_SFT
OUTNOT 1027.00  ; 3CH_OV/RN_NG_SFT_(取出)
; rung 21: CP1  NG
LD 720.01  ; 1CH_L_NO_(CP1)
@LD 701.00  ; ﾃﾞｰﾀ_ｼﾌﾄ
LD 701.05  ; ｼﾌﾄﾃﾞｰﾀ_ｸﾘｱ
SFT(010) 1031 1031  ; L_NO_(CP1)
; rung 22
LD 720.02  ; 1CH_R_NO_(CP1)
@LD 701.00  ; ﾃﾞｰﾀ_ｼﾌﾄ
LD 701.05  ; ｼﾌﾄﾃﾞｰﾀ_ｸﾘｱ
SFT(010) 1032 1032  ; R_NO_(CP1)

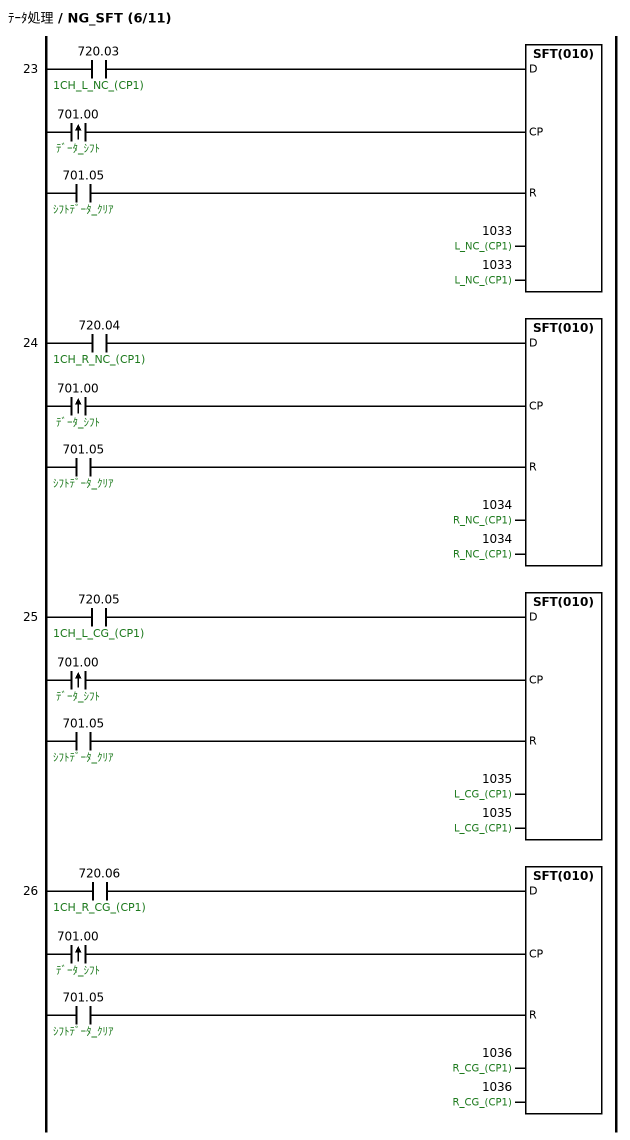
; rung 23
LD 720.03  ; 1CH_L_NC_(CP1)
@LD 701.00  ; ﾃﾞｰﾀ_ｼﾌﾄ
LD 701.05  ; ｼﾌﾄﾃﾞｰﾀ_ｸﾘｱ
SFT(010) 1033 1033  ; L_NC_(CP1)
; rung 24
LD 720.04  ; 1CH_R_NC_(CP1)
@LD 701.00  ; ﾃﾞｰﾀ_ｼﾌﾄ
LD 701.05  ; ｼﾌﾄﾃﾞｰﾀ_ｸﾘｱ
SFT(010) 1034 1034  ; R_NC_(CP1)
; rung 25
LD 720.05  ; 1CH_L_CG_(CP1)
@LD 701.00  ; ﾃﾞｰﾀ_ｼﾌﾄ
LD 701.05  ; ｼﾌﾄﾃﾞｰﾀ_ｸﾘｱ
SFT(010) 1035 1035  ; L_CG_(CP1)
; rung 26
LD 720.06  ; 1CH_R_CG_(CP1)
@LD 701.00  ; ﾃﾞｰﾀ_ｼﾌﾄ
LD 701.05  ; ｼﾌﾄﾃﾞｰﾀ_ｸﾘｱ
SFT(010) 1036 1036  ; R_CG_(CP1)

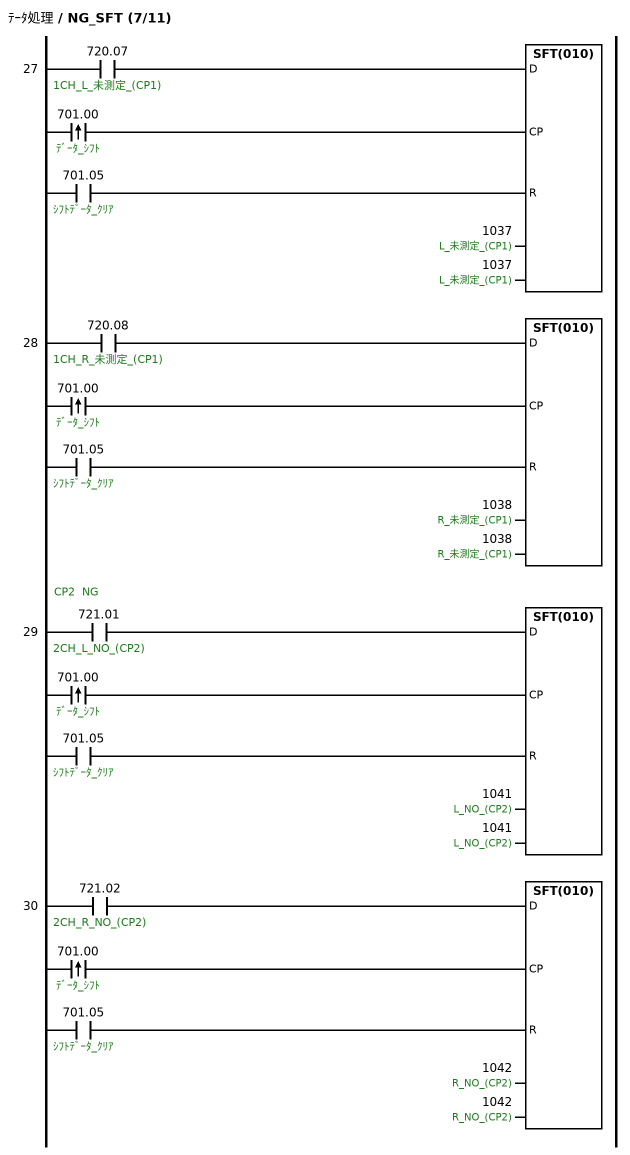
; rung 27
LD 720.07  ; 1CH_L_未測定_(CP1)
@LD 701.00  ; ﾃﾞｰﾀ_ｼﾌﾄ
LD 701.05  ; ｼﾌﾄﾃﾞｰﾀ_ｸﾘｱ
SFT(010) 1037 1037  ; L_未測定_(CP1)
; rung 28
LD 720.08  ; 1CH_R_未測定_(CP1)
@LD 701.00  ; ﾃﾞｰﾀ_ｼﾌﾄ
LD 701.05  ; ｼﾌﾄﾃﾞｰﾀ_ｸﾘｱ
SFT(010) 1038 1038  ; R_未測定_(CP1)
; rung 29: CP2  NG
LD 721.01  ; 2CH_L_NO_(CP2)
@LD 701.00  ; ﾃﾞｰﾀ_ｼﾌﾄ
LD 701.05  ; ｼﾌﾄﾃﾞｰﾀ_ｸﾘｱ
SFT(010) 1041 1041  ; L_NO_(CP2)
; rung 30
LD 721.02  ; 2CH_R_NO_(CP2)
@LD 701.00  ; ﾃﾞｰﾀ_ｼﾌﾄ
LD 701.05  ; ｼﾌﾄﾃﾞｰﾀ_ｸﾘｱ
SFT(010) 1042 1042  ; R_NO_(CP2)

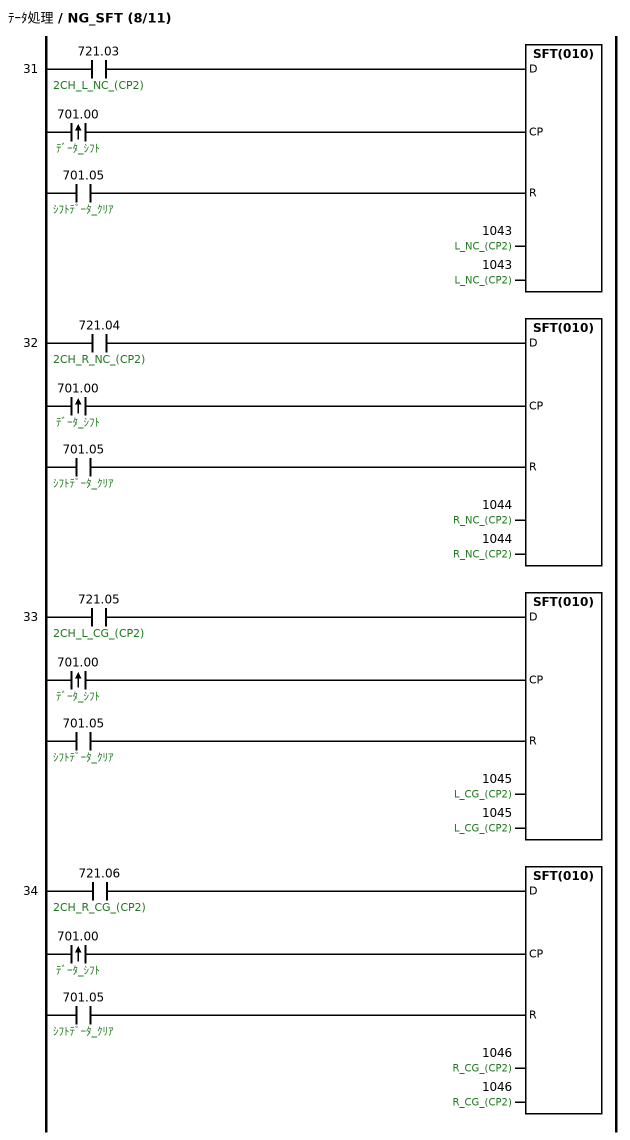
; rung 31
LD 721.03  ; 2CH_L_NC_(CP2)
@LD 701.00  ; ﾃﾞｰﾀ_ｼﾌﾄ
LD 701.05  ; ｼﾌﾄﾃﾞｰﾀ_ｸﾘｱ
SFT(010) 1043 1043  ; L_NC_(CP2)
; rung 32
LD 721.04  ; 2CH_R_NC_(CP2)
@LD 701.00  ; ﾃﾞｰﾀ_ｼﾌﾄ
LD 701.05  ; ｼﾌﾄﾃﾞｰﾀ_ｸﾘｱ
SFT(010) 1044 1044  ; R_NC_(CP2)
; rung 33
LD 721.05  ; 2CH_L_CG_(CP2)
@LD 701.00  ; ﾃﾞｰﾀ_ｼﾌﾄ
LD 701.05  ; ｼﾌﾄﾃﾞｰﾀ_ｸﾘｱ
SFT(010) 1045 1045  ; L_CG_(CP2)
; rung 34
LD 721.06  ; 2CH_R_CG_(CP2)
@LD 701.00  ; ﾃﾞｰﾀ_ｼﾌﾄ
LD 701.05  ; ｼﾌﾄﾃﾞｰﾀ_ｸﾘｱ
SFT(010) 1046 1046  ; R_CG_(CP2)

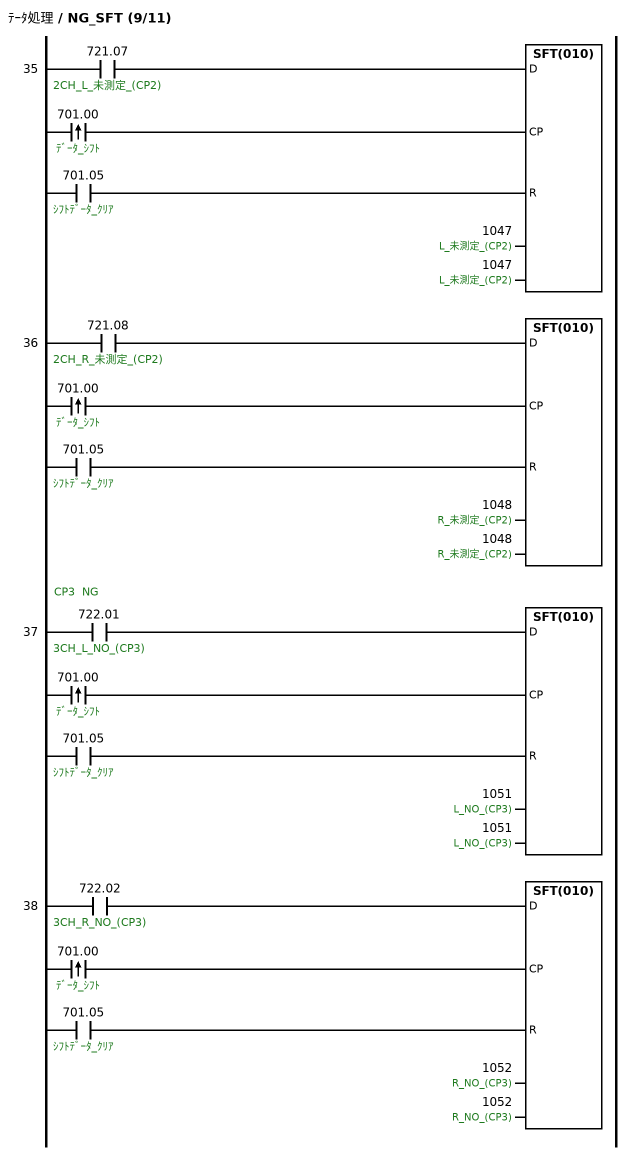
; rung 35
LD 721.07  ; 2CH_L_未測定_(CP2)
@LD 701.00  ; ﾃﾞｰﾀ_ｼﾌﾄ
LD 701.05  ; ｼﾌﾄﾃﾞｰﾀ_ｸﾘｱ
SFT(010) 1047 1047  ; L_未測定_(CP2)
; rung 36
LD 721.08  ; 2CH_R_未測定_(CP2)
@LD 701.00  ; ﾃﾞｰﾀ_ｼﾌﾄ
LD 701.05  ; ｼﾌﾄﾃﾞｰﾀ_ｸﾘｱ
SFT(010) 1048 1048  ; R_未測定_(CP2)
; rung 37: CP3  NG
LD 722.01  ; 3CH_L_NO_(CP3)
@LD 701.00  ; ﾃﾞｰﾀ_ｼﾌﾄ
LD 701.05  ; ｼﾌﾄﾃﾞｰﾀ_ｸﾘｱ
SFT(010) 1051 1051  ; L_NO_(CP3)
; rung 38
LD 722.02  ; 3CH_R_NO_(CP3)
@LD 701.00  ; ﾃﾞｰﾀ_ｼﾌﾄ
LD 701.05  ; ｼﾌﾄﾃﾞｰﾀ_ｸﾘｱ
SFT(010) 1052 1052  ; R_NO_(CP3)

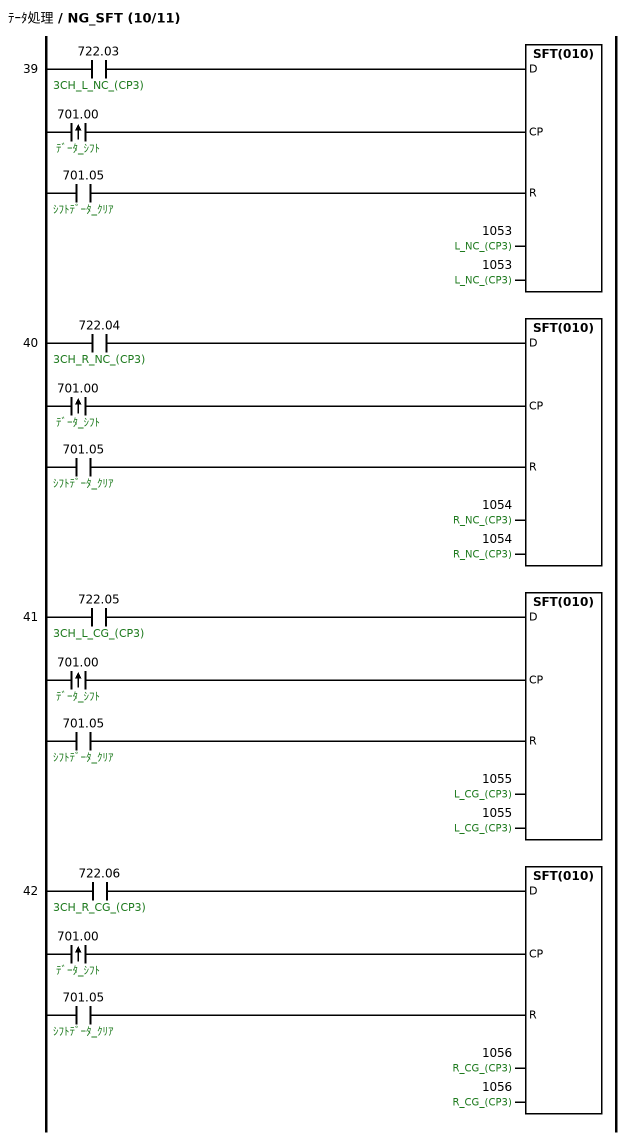
; rung 39
LD 722.03  ; 3CH_L_NC_(CP3)
@LD 701.00  ; ﾃﾞｰﾀ_ｼﾌﾄ
LD 701.05  ; ｼﾌﾄﾃﾞｰﾀ_ｸﾘｱ
SFT(010) 1053 1053  ; L_NC_(CP3)
; rung 40
LD 722.04  ; 3CH_R_NC_(CP3)
@LD 701.00  ; ﾃﾞｰﾀ_ｼﾌﾄ
LD 701.05  ; ｼﾌﾄﾃﾞｰﾀ_ｸﾘｱ
SFT(010) 1054 1054  ; R_NC_(CP3)
; rung 41
LD 722.05  ; 3CH_L_CG_(CP3)
@LD 701.00  ; ﾃﾞｰﾀ_ｼﾌﾄ
LD 701.05  ; ｼﾌﾄﾃﾞｰﾀ_ｸﾘｱ
SFT(010) 1055 1055  ; L_CG_(CP3)
; rung 42
LD 722.06  ; 3CH_R_CG_(CP3)
@LD 701.00  ; ﾃﾞｰﾀ_ｼﾌﾄ
LD 701.05  ; ｼﾌﾄﾃﾞｰﾀ_ｸﾘｱ
SFT(010) 1056 1056  ; R_CG_(CP3)

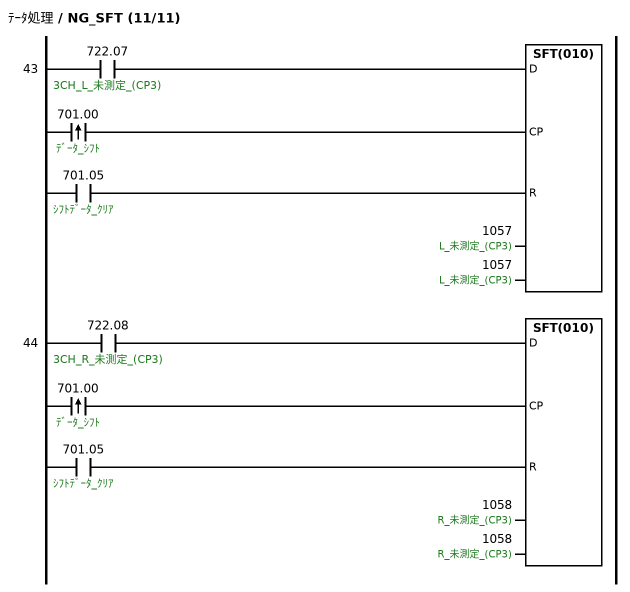
; rung 43
LD 722.07  ; 3CH_L_未測定_(CP3)
@LD 701.00  ; ﾃﾞｰﾀ_ｼﾌﾄ
LD 701.05  ; ｼﾌﾄﾃﾞｰﾀ_ｸﾘｱ
SFT(010) 1057 1057  ; L_未測定_(CP3)
; rung 44
LD 722.08  ; 3CH_R_未測定_(CP3)
@LD 701.00  ; ﾃﾞｰﾀ_ｼﾌﾄ
LD 701.05  ; ｼﾌﾄﾃﾞｰﾀ_ｸﾘｱ
SFT(010) 1058 1058  ; R_未測定_(CP3)

### Section OK_SFT

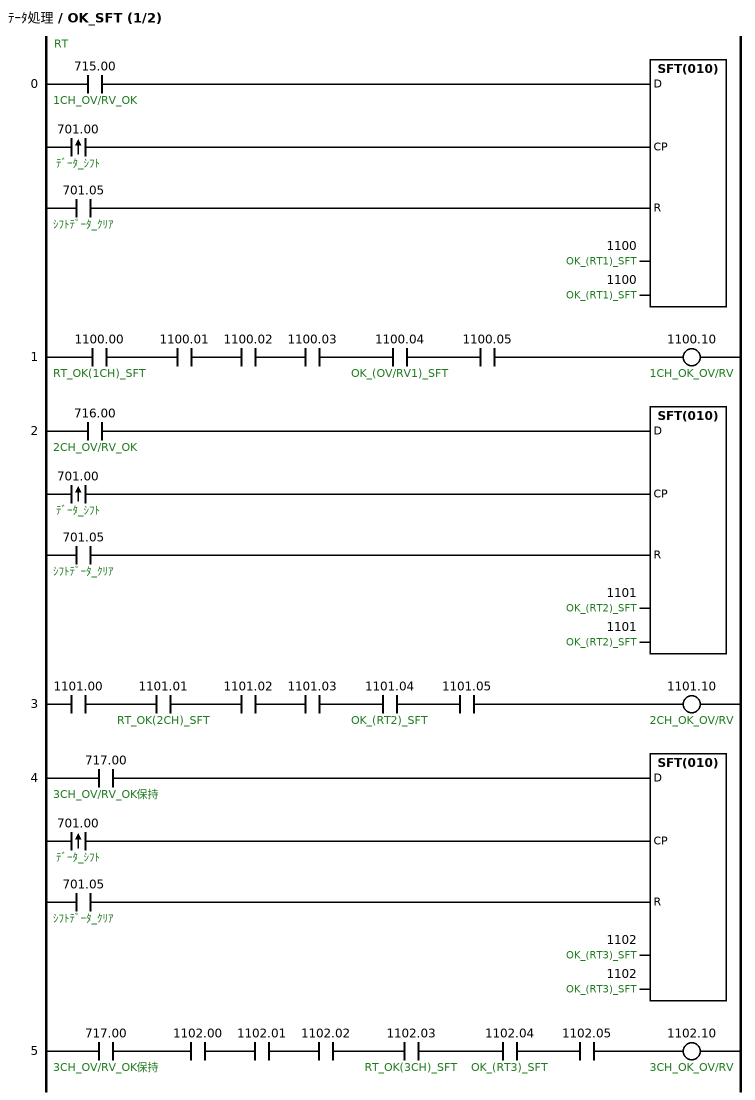
; rung 0: RT
LD 715.00  ; 1CH_OV/RV_OK
@LD 701.00  ; ﾃﾞｰﾀ_ｼﾌﾄ
LD 701.05  ; ｼﾌﾄﾃﾞｰﾀ_ｸﾘｱ
SFT(010) 1100 1100  ; OK_(RT1)_SFT
; rung 1
LD 1100.00  ; RT_OK(1CH)_SFT
AND 1100.01
AND 1100.02
AND 1100.03
AND 1100.04  ; OK_(OV/RV1)_SFT
AND 1100.05
OUT 1100.10  ; 1CH_OK_OV/RV
; rung 2
LD 716.00  ; 2CH_OV/RV_OK
@LD 701.00  ; ﾃﾞｰﾀ_ｼﾌﾄ
LD 701.05  ; ｼﾌﾄﾃﾞｰﾀ_ｸﾘｱ
SFT(010) 1101 1101  ; OK_(RT2)_SFT
; rung 3
LD 1101.00
AND 1101.01  ; RT_OK(2CH)_SFT
AND 1101.02
AND 1101.03
AND 1101.04  ; OK_(RT2)_SFT
AND 1101.05
OUT 1101.10  ; 2CH_OK_OV/RV
; rung 4
LD 717.00  ; 3CH_OV/RV_OK保持
@LD 701.00  ; ﾃﾞｰﾀ_ｼﾌﾄ
LD 701.05  ; ｼﾌﾄﾃﾞｰﾀ_ｸﾘｱ
SFT(010) 1102 1102  ; OK_(RT3)_SFT
; rung 5
LD 717.00  ; 3CH_OV/RV_OK保持
AND 1102.00
AND 1102.01
AND 1102.02
AND 1102.03  ; RT_OK(3CH)_SFT
AND 1102.04  ; OK_(RT3)_SFT
AND 1102.05
OUT 1102.10  ; 3CH_OK_OV/RV

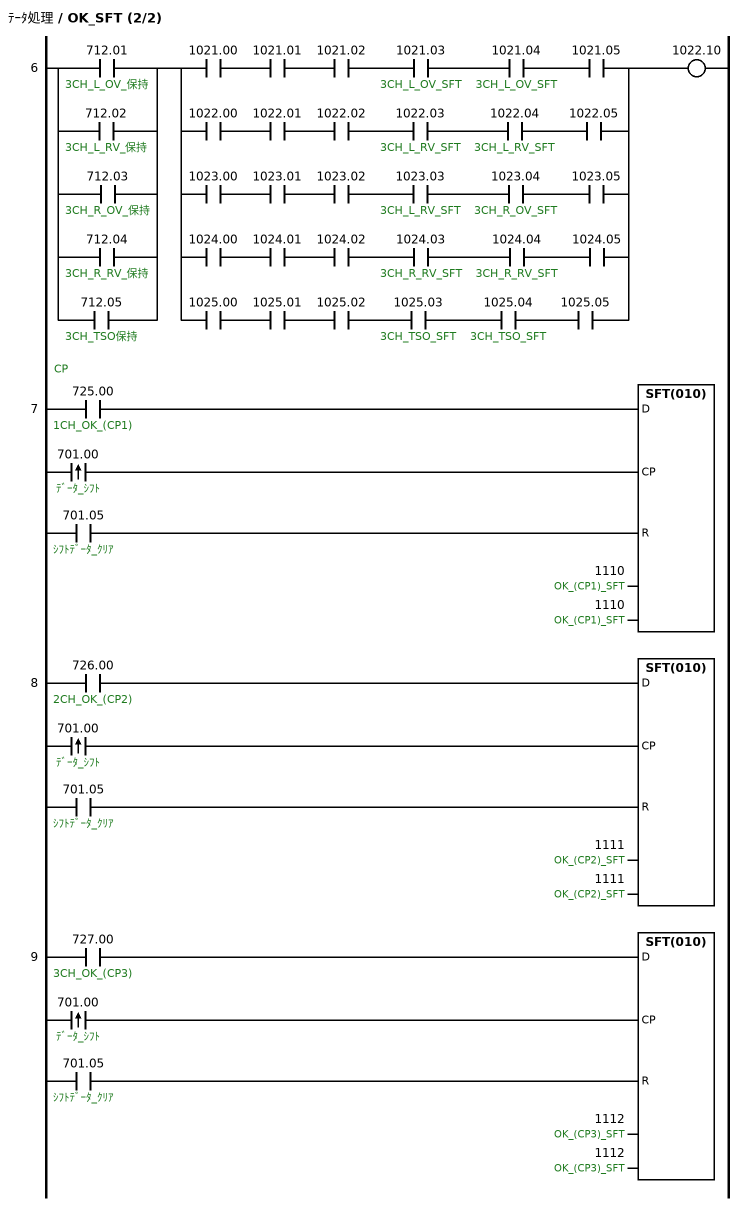
; rung 6
LD 712.01  ; 3CH_L_OV_保持
OR 712.02  ; 3CH_L_RV_保持
OR 712.03  ; 3CH_R_OV_保持
OR 712.04  ; 3CH_R_RV_保持
OR 712.05  ; 3CH_TSO保持
LD 1021.00
AND 1021.01
AND 1021.02
AND 1021.03  ; 3CH_L_OV_SFT
AND 1021.04  ; 3CH_L_OV_SFT
AND 1021.05
LD 1022.00
AND 1022.01
AND 1022.02
AND 1022.03  ; 3CH_L_RV_SFT
AND 1022.04  ; 3CH_L_RV_SFT
AND 1022.05
ORLD
LD 1023.00
AND 1023.01
AND 1023.02
AND 1023.03  ; 3CH_L_RV_SFT
AND 1023.04  ; 3CH_R_OV_SFT
AND 1023.05
ORLD
LD 1024.00
AND 1024.01
AND 1024.02
AND 1024.03  ; 3CH_R_RV_SFT
AND 1024.04  ; 3CH_R_RV_SFT
AND 1024.05
ORLD
LD 1025.00
AND 1025.01
AND 1025.02
AND 1025.03  ; 3CH_TSO_SFT
AND 1025.04  ; 3CH_TSO_SFT
AND 1025.05
ORLD
ANDLD
OUT 1022.10
; rung 7: CP
LD 725.00  ; 1CH_OK_(CP1)
@LD 701.00  ; ﾃﾞｰﾀ_ｼﾌﾄ
LD 701.05  ; ｼﾌﾄﾃﾞｰﾀ_ｸﾘｱ
SFT(010) 1110 1110  ; OK_(CP1)_SFT
; rung 8
LD 726.00  ; 2CH_OK_(CP2)
@LD 701.00  ; ﾃﾞｰﾀ_ｼﾌﾄ
LD 701.05  ; ｼﾌﾄﾃﾞｰﾀ_ｸﾘｱ
SFT(010) 1111 1111  ; OK_(CP2)_SFT
; rung 9
LD 727.00  ; 3CH_OK_(CP3)
@LD 701.00  ; ﾃﾞｰﾀ_ｼﾌﾄ
LD 701.05  ; ｼﾌﾄﾃﾞｰﾀ_ｸﾘｱ
SFT(010) 1112 1112  ; OK_(CP3)_SFT

### Section ﾃﾞｰﾀ処理

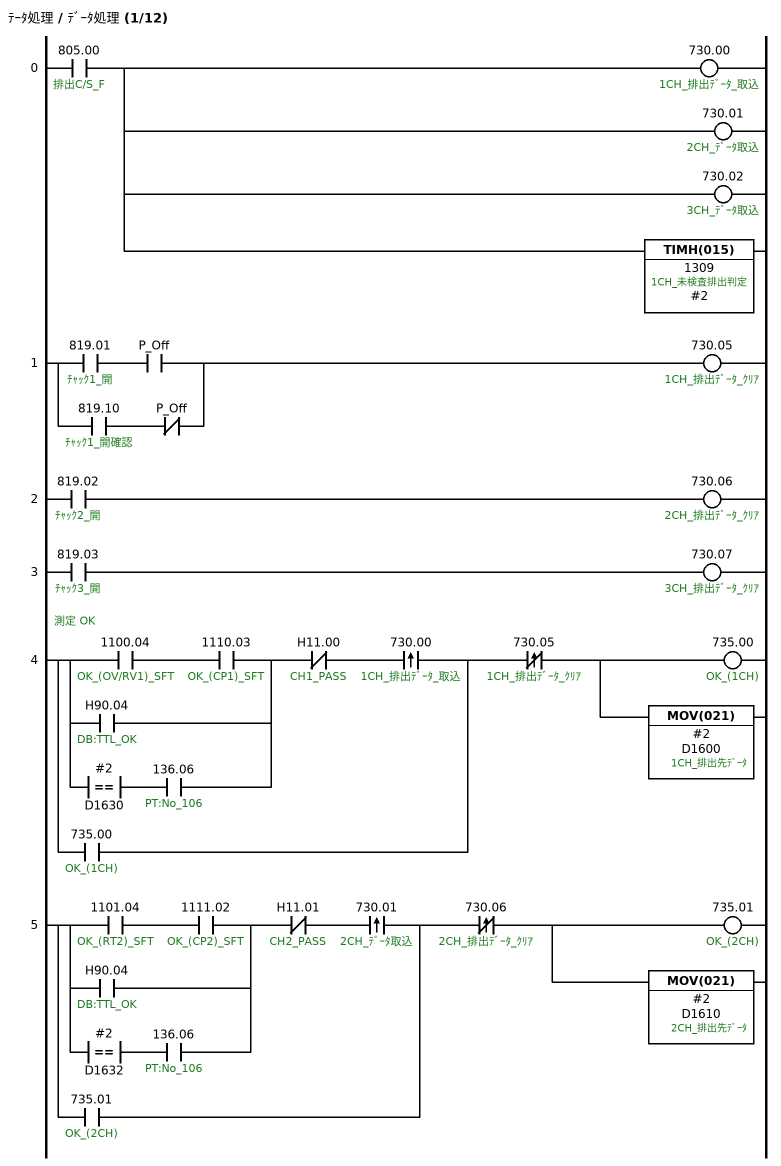
; rung 0
LD 805.00  ; 排出C/S_F
OUT 730.00  ; 1CH_排出ﾃﾞｰﾀ_取込
OUT 730.01  ; 2CH_ﾃﾞｰﾀ取込
OUT 730.02  ; 3CH_ﾃﾞｰﾀ取込
TIMH(015) 1309 #2  ; 1CH_未検査排出判定
; rung 1
LD 819.01  ; ﾁｬｯｸ1_開
AND P_Off
LD 819.10  ; ﾁｬｯｸ1_開確認
ANDNOT P_Off
ORLD
OUT 730.05  ; 1CH_排出ﾃﾞｰﾀ_ｸﾘｱ
; rung 2
LD 819.02  ; ﾁｬｯｸ2_開
OUT 730.06  ; 2CH_排出ﾃﾞｰﾀ_ｸﾘｱ
; rung 3
LD 819.03  ; ﾁｬｯｸ3_開
OUT 730.07  ; 3CH_排出ﾃﾞｰﾀ_ｸﾘｱ
; rung 4: 測定 OK
LD 1100.04  ; OK_(OV/RV1)_SFT
AND 1110.03  ; OK_(CP1)_SFT
OR H90.04  ; DB:TTL_OK
LD=(300) #2 D1630
AND 136.06  ; PT:No_106
ORLD
ANDNOT H11.00  ; CH1_PASS
@AND 730.00  ; 1CH_排出ﾃﾞｰﾀ_取込
OR 735.00  ; OK_(1CH)
@ANDNOT 730.05  ; 1CH_排出ﾃﾞｰﾀ_ｸﾘｱ
OUT 735.00  ; OK_(1CH)
MOV(021) #2 D1600  ; 1CH_排出先ﾃﾞｰﾀ
; rung 5
LD 1101.04  ; OK_(RT2)_SFT
AND 1111.02  ; OK_(CP2)_SFT
OR H90.04  ; DB:TTL_OK
LD=(300) #2 D1632
AND 136.06  ; PT:No_106
ORLD
ANDNOT H11.01  ; CH2_PASS
@AND 730.01  ; 2CH_ﾃﾞｰﾀ取込
OR 735.01  ; OK_(2CH)
@ANDNOT 730.06  ; 2CH_排出ﾃﾞｰﾀ_ｸﾘｱ
OUT 735.01  ; OK_(2CH)
MOV(021) #2 D1610  ; 2CH_排出先ﾃﾞｰﾀ

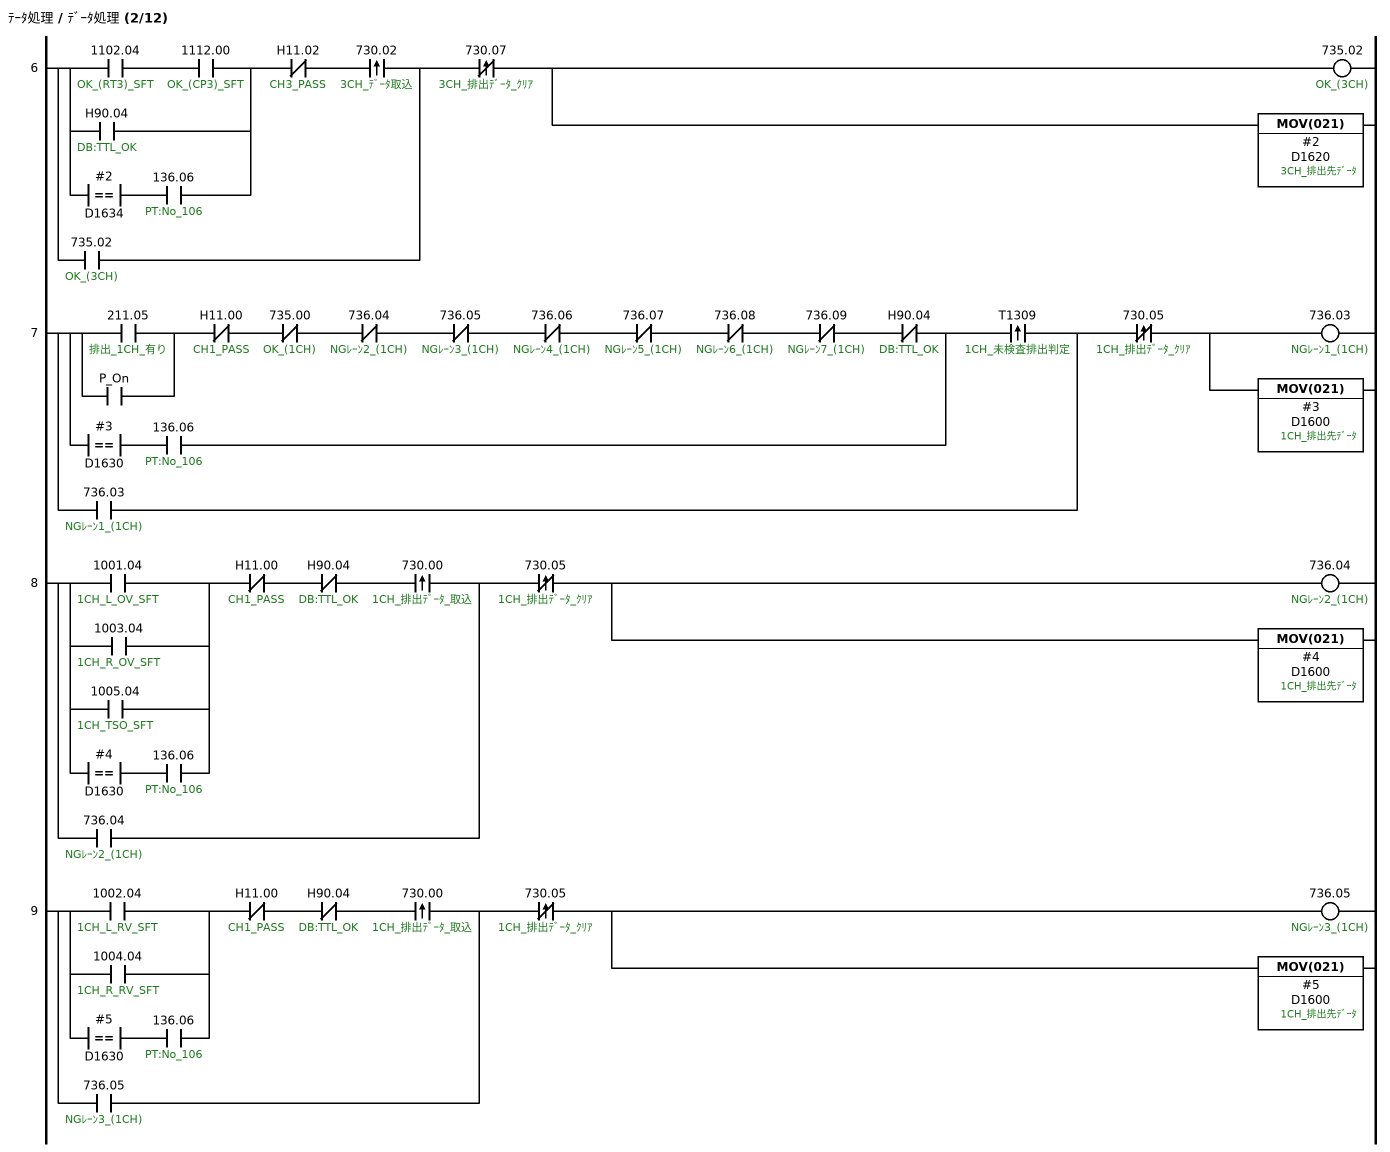
; rung 6
LD 1102.04  ; OK_(RT3)_SFT
AND 1112.00  ; OK_(CP3)_SFT
OR H90.04  ; DB:TTL_OK
LD=(300) #2 D1634
AND 136.06  ; PT:No_106
ORLD
ANDNOT H11.02  ; CH3_PASS
@AND 730.02  ; 3CH_ﾃﾞｰﾀ取込
OR 735.02  ; OK_(3CH)
@ANDNOT 730.07  ; 3CH_排出ﾃﾞｰﾀ_ｸﾘｱ
OUT 735.02  ; OK_(3CH)
MOV(021) #2 D1620  ; 3CH_排出先ﾃﾞｰﾀ
; rung 7
LD 211.05  ; 排出_1CH_有り
OR P_On
ANDNOT H11.00  ; CH1_PASS
ANDNOT 735.00  ; OK_(1CH)
ANDNOT 736.04  ; NGﾚｰﾝ2_(1CH)
ANDNOT 736.05  ; NGﾚｰﾝ3_(1CH)
ANDNOT 736.06  ; NGﾚｰﾝ4_(1CH)
ANDNOT 736.07  ; NGﾚｰﾝ5_(1CH)
ANDNOT 736.08  ; NGﾚｰﾝ6_(1CH)
ANDNOT 736.09  ; NGﾚｰﾝ7_(1CH)
ANDNOT H90.04  ; DB:TTL_OK
LD=(300) #3 D1630
AND 136.06  ; PT:No_106
ORLD
@AND T1309  ; 1CH_未検査排出判定
OR 736.03  ; NGﾚｰﾝ1_(1CH)
@ANDNOT 730.05  ; 1CH_排出ﾃﾞｰﾀ_ｸﾘｱ
OUT 736.03  ; NGﾚｰﾝ1_(1CH)
MOV(021) #3 D1600  ; 1CH_排出先ﾃﾞｰﾀ
; rung 8
LD 1001.04  ; 1CH_L_OV_SFT
OR 1003.04  ; 1CH_R_OV_SFT
OR 1005.04  ; 1CH_TSO_SFT
LD=(300) #4 D1630
AND 136.06  ; PT:No_106
ORLD
ANDNOT H11.00  ; CH1_PASS
ANDNOT H90.04  ; DB:TTL_OK
@AND 730.00  ; 1CH_排出ﾃﾞｰﾀ_取込
OR 736.04  ; NGﾚｰﾝ2_(1CH)
@ANDNOT 730.05  ; 1CH_排出ﾃﾞｰﾀ_ｸﾘｱ
OUT 736.04  ; NGﾚｰﾝ2_(1CH)
MOV(021) #4 D1600  ; 1CH_排出先ﾃﾞｰﾀ
; rung 9
LD 1002.04  ; 1CH_L_RV_SFT
OR 1004.04  ; 1CH_R_RV_SFT
LD=(300) #5 D1630
AND 136.06  ; PT:No_106
ORLD
ANDNOT H11.00  ; CH1_PASS
ANDNOT H90.04  ; DB:TTL_OK
@AND 730.00  ; 1CH_排出ﾃﾞｰﾀ_取込
OR 736.05  ; NGﾚｰﾝ3_(1CH)
@ANDNOT 730.05  ; 1CH_排出ﾃﾞｰﾀ_ｸﾘｱ
OUT 736.05  ; NGﾚｰﾝ3_(1CH)
MOV(021) #5 D1600  ; 1CH_排出先ﾃﾞｰﾀ

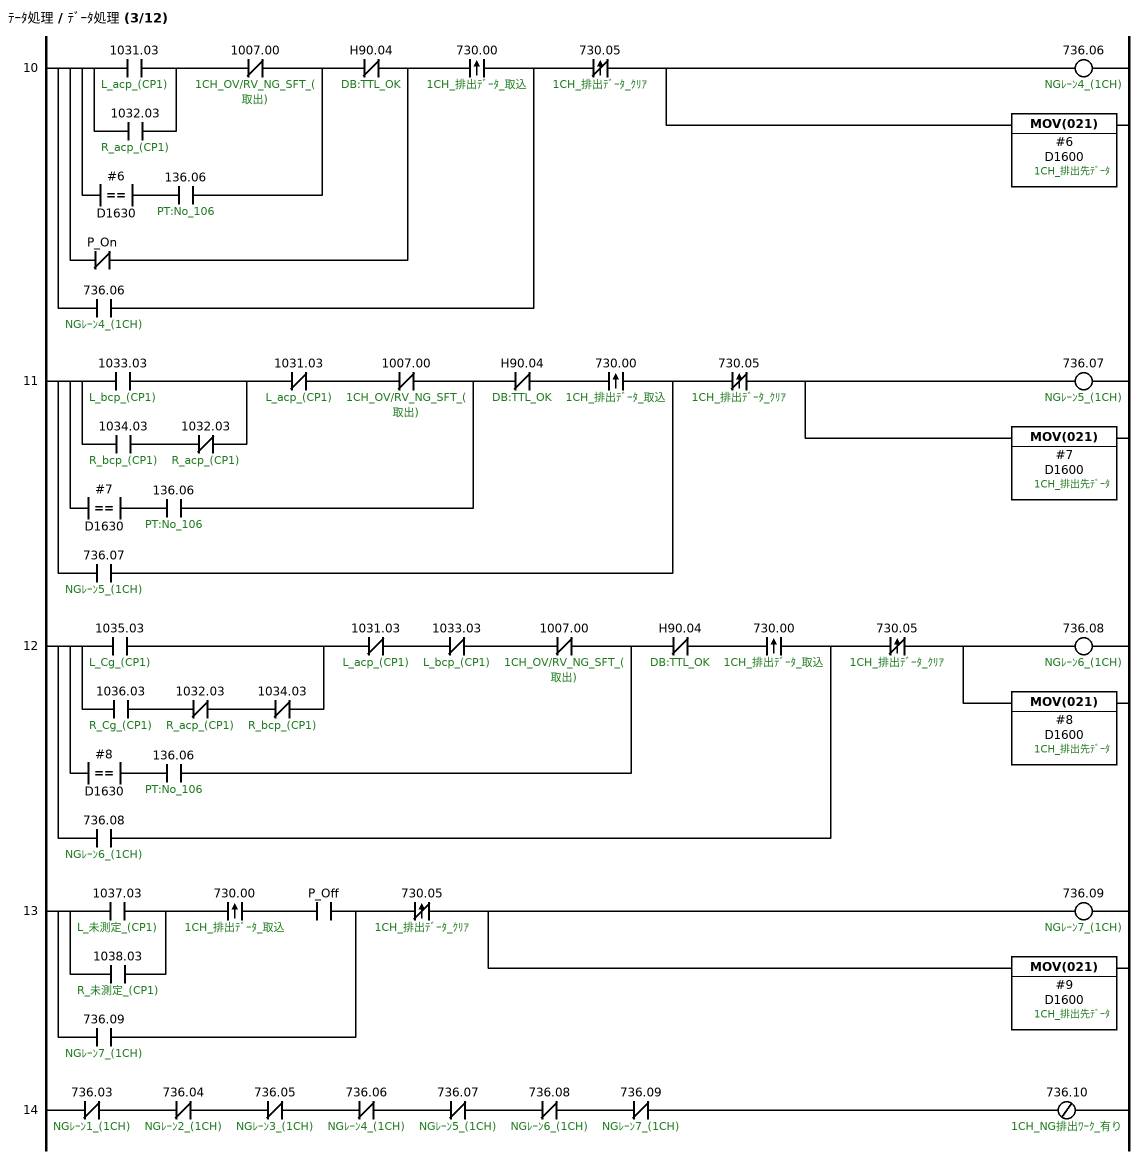
; rung 10
LD 1031.03  ; L_acp_(CP1)
OR 1032.03  ; R_acp_(CP1)
ANDNOT 1007.00  ; 1CH_OV/RV_NG_SFT_(取出)
LD=(300) #6 D1630
AND 136.06  ; PT:No_106
ORLD
ANDNOT H90.04  ; DB:TTL_OK
ORNOT P_On
@AND 730.00  ; 1CH_排出ﾃﾞｰﾀ_取込
OR 736.06  ; NGﾚｰﾝ4_(1CH)
@ANDNOT 730.05  ; 1CH_排出ﾃﾞｰﾀ_ｸﾘｱ
OUT 736.06  ; NGﾚｰﾝ4_(1CH)
MOV(021) #6 D1600  ; 1CH_排出先ﾃﾞｰﾀ
; rung 11
LD 1033.03  ; L_bcp_(CP1)
LD 1034.03  ; R_bcp_(CP1)
ANDNOT 1032.03  ; R_acp_(CP1)
ORLD
ANDNOT 1031.03  ; L_acp_(CP1)
ANDNOT 1007.00  ; 1CH_OV/RV_NG_SFT_(取出)
LD=(300) #7 D1630
AND 136.06  ; PT:No_106
ORLD
ANDNOT H90.04  ; DB:TTL_OK
@AND 730.00  ; 1CH_排出ﾃﾞｰﾀ_取込
OR 736.07  ; NGﾚｰﾝ5_(1CH)
@ANDNOT 730.05  ; 1CH_排出ﾃﾞｰﾀ_ｸﾘｱ
OUT 736.07  ; NGﾚｰﾝ5_(1CH)
MOV(021) #7 D1600  ; 1CH_排出先ﾃﾞｰﾀ
; rung 12
LD 1035.03  ; L_Cg_(CP1)
LD 1036.03  ; R_Cg_(CP1)
ANDNOT 1032.03  ; R_acp_(CP1)
ANDNOT 1034.03  ; R_bcp_(CP1)
ORLD
ANDNOT 1031.03  ; L_acp_(CP1)
ANDNOT 1033.03  ; L_bcp_(CP1)
ANDNOT 1007.00  ; 1CH_OV/RV_NG_SFT_(取出)
LD=(300) #8 D1630
AND 136.06  ; PT:No_106
ORLD
ANDNOT H90.04  ; DB:TTL_OK
@AND 730.00  ; 1CH_排出ﾃﾞｰﾀ_取込
OR 736.08  ; NGﾚｰﾝ6_(1CH)
@ANDNOT 730.05  ; 1CH_排出ﾃﾞｰﾀ_ｸﾘｱ
OUT 736.08  ; NGﾚｰﾝ6_(1CH)
MOV(021) #8 D1600  ; 1CH_排出先ﾃﾞｰﾀ
; rung 13
LD 1037.03  ; L_未測定_(CP1)
OR 1038.03  ; R_未測定_(CP1)
@AND 730.00  ; 1CH_排出ﾃﾞｰﾀ_取込
AND P_Off
OR 736.09  ; NGﾚｰﾝ7_(1CH)
@ANDNOT 730.05  ; 1CH_排出ﾃﾞｰﾀ_ｸﾘｱ
OUT 736.09  ; NGﾚｰﾝ7_(1CH)
MOV(021) #9 D1600  ; 1CH_排出先ﾃﾞｰﾀ
; rung 14
LDNOT 736.03  ; NGﾚｰﾝ1_(1CH)
ANDNOT 736.04  ; NGﾚｰﾝ2_(1CH)
ANDNOT 736.05  ; NGﾚｰﾝ3_(1CH)
ANDNOT 736.06  ; NGﾚｰﾝ4_(1CH)
ANDNOT 736.07  ; NGﾚｰﾝ5_(1CH)
ANDNOT 736.08  ; NGﾚｰﾝ6_(1CH)
ANDNOT 736.09  ; NGﾚｰﾝ7_(1CH)
OUTNOT 736.10  ; 1CH_NG排出ﾜｰｸ_有り

